# B&R Automation Studio project Parker_BMM_ST_V5_3147_V12 (part 8)

```c
		case 22000:
			pMold->Clamp.vRamp.Ts = tTask;
			pMold->Clamp.vRamp.Set = 0.0;

			/* call profile function */
			HydSCurveRamp(&pMold->Clamp.vRamp);

			pMold->Clamp.p_set = pMold->Clamp.p_old;
			pMold->Clamp.v_set = pMold->Clamp.vRamp.Out;

			if(pMold->Clamp.v_set < 0.1 && pMold->Clamp.v_set > -0.1)
			{
				pMold->Clamp.v_set = 0.0;
				pMold->Clamp.p_set =0;
				pMold->Clamp.Step = 0;
			}
			break;

		/* ----------------------------  Instance stop ------------------------- */
		case 30000:
			pMold->Clamp.Timer.IN      = 0;
			pMold->Clamp.LimitTimer.IN = 0;
			pMoldUser->Clamp.Timer.IN = 0;/*Albert*/

			pMold->ActInfo.ClampOpn = 0;
			pMold->ActInfo.ClampCls = 0;

			//*--VALVE_DIR--*//
			/*-- Close --*/
			pMold->ValveOut.ClampCls  = 0;
			pMold->ValveOut.ClampClsDiff = 0;
			pMold->ValveOut.ClampClsSlow = 0;
			/*-- Close_Tonnage_additional --*/
			pMold->ValveOut.Lock = 0;
			pMold->ValveOut.ClampClsAux = 0;

			/*-- Open --*/
			pMold->ValveOut.ClampOpn  = 0;
			pMold->ValveOut.ClampOpnDiff = 0;
			pMold->ValveOut.ClampOpnRelease = 0;

			//*--VALVE_PROP--*//
			pMold->ValveOut.ClampMoveValve = 0;

			/*-- Close --*/
			pMold->ValveOut.ClampClsDiff = 0;
			pMold->ValveOut.ClampClsSlow = 0;

			/*-- Open --*/
			pMold->ValveOut.ClampOpnDiff = 0;
			pMold->ValveOut.ClampOpnRelease = 0;

			pMold->Clamp.vRamp.Once = 0;
			pMold->Clamp.vRamp.Set = pMold->Clamp.v_set;

			pMold->Clamp.vRamp.Ts = tTask;

			pMold->Clamp.vRamp.Accel = INSTANCY_STOP_ACCEL;

			/* call profile function */
			HydSCurveRamp(&pMold->Clamp.vRamp);

			//	pMold->Clamp.p_set = 100.0;
			pMold->Clamp.v_set = pMold->Clamp.vRamp.Out;

			pMold->Clamp.Step = 31000;
			break;

		case 31000:
			pMold->Clamp.vRamp.Ts = tTask;
			pMold->Clamp.vRamp.Set = 0.0;

			/* call profile function */
			HydSCurveRamp(&pMold->Clamp.vRamp);

			pMold->Clamp.p_set = pMold->Clamp.p_old;
			pMold->Clamp.v_set = pMold->Clamp.vRamp.Out;

			if(pMold->Clamp.v_set < 0.1 && pMold->Clamp.v_set > -0.1)
			{
				pMold->Clamp.v_set = 0.0;
				pMold->Clamp.p_set =0;
				pMold->Clamp.Step = 0;
			}
			break;

		/* ----------------------------  Error step ------------------------- */
		case 40000:
			pMold->Clamp.Timer.IN      = 0;
			pMold->Clamp.LimitTimer.IN = 0;

			pMold->ActInfo.ClampOpn = 0;
			pMold->ActInfo.ClampCls = 0;

			pMold->Clamp.v_set = 0.0;
			pMold->Clamp.p_set =0;

			//*--VALVE_DIR--*//
			/*-- Close --*/
			pMold->ValveOut.ClampCls  = 0;
			pMold->ValveOut.ClampClsDiff = 0;
			pMold->ValveOut.ClampClsSlow = 0;
			/*-- Close_Tonnage_additional --*/
			pMold->ValveOut.Lock = 0;
			pMold->ValveOut.ClampClsAux = 0;

			/*-- Open --*/
			pMold->ValveOut.ClampOpn  = 0;
			pMold->ValveOut.ClampOpnDiff = 0;
			pMold->ValveOut.ClampOpnRelease = 0;

			//*--VALVE_PROP--*//
			pMold->ValveOut.ClampMoveValve = 0;

			/*-- Close --*/
			pMold->ValveOut.ClampClsDiff = 0;
			pMold->ValveOut.ClampClsSlow = 0;

			/*-- Open --*/
			pMold->ValveOut.ClampOpnDiff = 0;
			pMold->ValveOut.ClampOpnRelease = 0;

			break;

		/* ----------------------------  auto run stop ------------------------- */
		case 41000:
			pMold->Clamp.Timer.IN      = 0;
			pMold->Clamp.LimitTimer.IN = 0;

			pMold->ActInfo.ClampOpn = 0;
			pMold->ActInfo.ClampCls = 0;

			pMold->Clamp.Step = 42000;
			break;

		case 42000:
			pMold->Clamp.vRamp.Internal.Once = 0;
			pMold->Clamp.vRamp.Set = pMold->Clamp.v_set;

			pMold->Clamp.vRamp.Ts = tTask;

			pMold->Clamp.vRamp.Accel = INSTANCY_STOP_ACCEL;

			/* call profile function */
			HydSCurveRamp(&pMold->Clamp.vRamp);
			pMold->Clamp.Step = 43000;
			break;

		case 43000:
			pMold->Clamp.vRamp.Ts = tTask;
			pMold->Clamp.vRamp.Set = 0.0;

			/* call profile function */
			HydSCurveRamp(&pMold->Clamp.vRamp);

			//	pMold->Clamp.p_set = 100.0;
			pMold->Clamp.v_set = pMold->Clamp.vRamp.Out;

			if(pMold->Clamp.v_set < 0.1 && pMold->Clamp.v_set > -0.1)
			{
				pMold->Clamp.p_set =0;
				pMold->Clamp.v_set = 0.0;
				pMold->Clamp.Step = 40000;
			}
			break;
	}/* end of switch */

	if(pMold->Clamp.Step > 300 && pMold->Clamp.Step  < 800)
	{
		pMold->TimeDis.ClampClsAlarmTime = pMold->Clamp.LimitTimer.ET;
	}
	else if(pMold->Clamp.Step > 10300 && pMold->Clamp.Step  < 10800)
	{
		pMold->TimeDis.ClampOpnAlarmTime = pMold->Clamp.LimitTimer.ET;
	}

	/* ----------------- clamp open / close timeout --------------------  */
	if(1 == pMold->Clamp.LimitTimer.Q && 1 == gMachineInfo.TimeLimit)
	{
		if(pMold->Clamp.Step < 4000 && pMold->Clamp.Step > 200)		/* clamp close  */
		{
			pMold->Alarm.ClampNotAtClsDI = 1;
		}

		if(pMold->Clamp.Step < 13000 && pMold->Clamp.Step > 10200)	/* clamp open  */
		{
			pMold->Alarm.ClampNotAtOpnDI = 1;
		}

		pMold->Clamp.LimitTimer.IN = 0;
		pMold->Clamp.Step = 41000;
	}

	/* ----------------- clamp open / close action limit --------------------  */

	if(pMold->Clamp.Step < 3000 && pMold->Clamp.Step > 200) 	/* clamp close  */
	{

		if( 0 == pMold->TransDIn.SubMoldClsLimit)
		{
			pMold->Alarm.SubMoldNotAtOpnPos  = !pMold->TransDIn.SubMoldOpnLimit;
			pMold->Clamp.Step = 41000;
		}

		if( 0 == pMold->TransDIn.BottomSubMoldClsLimit)
		{
			pMold->Alarm.SubMoldNotAtOpnPos  = !pMold->TransDIn.BottomSubMoldClsLimit;
			pMold->Clamp.Step = 41000;
		}

		if(1 == gMachineInfo.Auto && 1 == gMachineFix.Option.bCoolPinUpNextCycClampCls)   /* 特殊模式  "於下一循環關模後轉一上"  */
		{
			//			if ( 0 == pMold->TransDIn.CoolPin2UpLimit || 0 == pMold->TransDIn.CoolPin3UpLimit )
			//			{
			//				pMold->Alarm.CoolPin2NotAtUpPos = !pMold->TransDIn.CoolPin2UpLimit;
			//				pMold->Alarm.CoolPin3NotAtUpPos	= !pMold->TransDIn.CoolPin3UpLimit;
			//				pMold->Clamp.Step = 41000;
			//			}
		}
		else
		{
			if (0 == pMold->TransDIn.CoolPinUpLimit )
			{
				pMold->Alarm.CoolPinNotAtUpPos	= !pMold->TransDIn.CoolPinUpLimit;
				pMold->Clamp.Step = 41000;
			}

		}

		if(0 == gMachineInfo.Auto)
		{
			if(0 == pMold->Robot.Transfer.BwPos)
			{
				pMold->Alarm.RobotNotAtBwPos = !pMold->Robot.Transfer.BwPos;
				pMold->Clamp.Step = 41000;
			}
		}

		if(1 == gMachineInfo.Auto )
		{
			if(0 == pMold->Carriage.FwPos)
			{
				pMold->Alarm.CarriageNotAtFwDI  = !pMold->Carriage.FwPos;
				pMold->Clamp.Step = 41000;
			}
		}

		/* 模内吹针在回位   */
		//      if(0 == pMold->TransDIn.InnerPinBwLimit)
		//      {
		//         pMold->Alarm.InnerPinNotAtBwPos = !pMold->TransDIn.InnerPinBwLimit;
		//         pMold->Clamp.Step = 41000;
		//      }

		//      if(1 == gMachineInfo.TimeLimit)
		//      {
		//         if(0 == pMold->Carriage.FwPos)
		//         {
		//            pMold->Alarm.CarriageNotAtFwDI  = !pMold->Carriage.FwPos;
		//            pMold->Clamp.Step = 41000;
		//         }
		//      }
		//      else
		//      {
		//         if(0 == pMold->Carriage.BwPos
		//			&& 0 == pMold->Carriage.FwPos
		//			&& 0 == pMold->BlowPin.UpPos)
		//         {
		//         	pMold->Alarm.CarriageNotAtBwDI = !pMold->Carriage.BwPos;
		//         	pMold->Alarm.BlowPinNotAtUpPos = !pMold->BlowPin.UpPos;
		//         	pMold->Clamp.Step = 41000;
		//         }
		//      }/* if(1 == gMachineInfo.Manual) */
	}/* if(pMold->Clamp.Step < 3000 && pMold->Clamp.Step > 200) */

	if(pMold->Clamp.Step < 13000 && pMold->Clamp.Step > 10200)  /* clamp open  */
	{

		/* 切飞边非退位  */
		if( 0 == pMold->TransDIn.TopDeflashBwLimit )
		{
			pMold->Alarm.TopDeflashNotAtBwPos = !pMold->TransDIn.TopDeflashBwLimit;
			pMold->Clamp.Step = 41000;
		}

		if( 0 == pMold->TransDIn.BottomDeflashBwLimit)
		{
			pMold->Alarm.BottomDeflashNotAtBwPos = !pMold->TransDIn.BottomDeflashBwLimit;
			pMold->Clamp.Step = 41000;
		}

		if(0 == gMachineInfo.Auto)
		{
			if(0 == pMold->TransDIn.ExtRobotUpLmit )
			{
				pMold->Alarm.ExtRobotNotAtUp = !pMold->TransDIn.ExtRobotUpLmit;
				pMold->Clamp.Step = 41000;
			}
		}

	}/* if(pMold->Clamp.Step < 13000 && pMold->Clamp.Step > 10200) */

	//	if((13000 >= pMold->Clamp.Step) && (10200 < pMold->Clamp.Step))
	//	{
	//		if(pMold == &RMold)
	//		{
	//			RobotClampTime.IN = pMold->Clamp.OpnPos;/*Albert RobotClampOpn*/
	//			RobotClampTime.PT = RobotClampTimePara;
	//		}
	//		if(pMold == & LMold)
	//		{
	//			LRobotClampTime.IN = pMold->Clamp.OpnPos;
	//			LRobotClampTime.PT = LRobotClampTimePara;
	//		}
	//	}
	//	else
	//	{
	////		RobotClampTime.IN = 0;/*Albert RobotClampOpn*/
	//	}
	//	if(pMold == &RMold)
	//	{
	//		if(RobotClampTime.Q)
	//		{
	//			RobotClampTime.IN = 0;
	//		}
	//		pMold->ValveOut.RobotClampOpn = RobotClampTime.Q;
	//
	//	}
	//	if(pMold == &LMold)
	//	{
	//		if(LRobotClampTime.Q)
	//		{
	//			LRobotClampTime.IN = 0;
	//		}
	//		pMold->ValveOut.RobotClampOpn = LRobotClampTime.Q;
	//	}

	/* ------------------------------------------------------------------------------ */
	/* ----------------- clamp output and proportional valve linear  ---------------- */
	/* ------------------------------------------------------------------------------ */

	if (pClampFix->eValveType == VALVE_PROP)
	{
		if(bClampPropValveOutputInverse == 0 )
		{
			if((pClampFix->Open.VoltageMax - pClampFix->Open.VoltageMin > 5.0) &&
				(pClampFix->Close.VoltageMin - pClampFix->Close.VoltageMax > 5.0))
			{
				pMold->Clamp.PropValveOk   = 1;
				pMold->Alarm.ClampValveErr = 0;
			}
			else
			{
				pMold->Clamp.PropValveOk   = 0;
				pMold->Alarm.ClampValveErr = 1;
			}
		}
		else
		{
			if((pClampFix->Open.VoltageMin - pClampFix->Open.VoltageMax > 5.0) &&
				(pClampFix->Close.VoltageMax - pClampFix->Close.VoltageMin > 5.0))
			{
				pMold->Clamp.PropValveOk   = 1;
				pMold->Alarm.ClampValveErr = 0;
			}
			else
			{
				pMold->Clamp.PropValveOk   = 0;
				pMold->Alarm.ClampValveErr = 1;
			}
		}

		pClampFix->Close.V_Max = 1000;
		pClampFix->Open.V_Max  = 1000;

		if(pMold->Clamp.v_set > pClampFix->Open.V_Max) pMold->Clamp.v_set = pClampFix->Open.V_Max;
		if(pMold->Clamp.v_set < -pClampFix->Close.V_Max) pMold->Clamp.v_set = -pClampFix->Close.V_Max;

		if(5000 == pMold->Clamp.Step || 15000 == pMold->Clamp.Step || 8500 == pMold->Clamp.Step)
		{
			if(bClampPropValveOutputInverse == 0)
			{
				pMold->Clamp.aoPropValve = pMold->Clamp.v_set * 32767/100;   /* 电压输出  0 -- 100 ---> 0.0 -- 10.0v*/
			}
			else
			{
				pMold->Clamp.aoPropValve = -(pMold->Clamp.v_set * 32767/100);   /* 电压输出  0 -- 100 ---> 0.0 -- 10.0v*/
			}

		}
		else
		{
			if(pMold->Clamp.v_set > 0 && pMold->Clamp.v_set <= pClampFix->Open.V_Max)
			{
				if(bClampPropValveOutputInverse == 0)
				{
					//Open +V
					pMold->Clamp.aoPropValve = 3276 * (pClampFix->Open.VoltageMin + pMold->Clamp.v_set/pClampFix->Open.V_Max *
						(pClampFix->Open.VoltageMax - pClampFix->Open.VoltageMin));
				}
				else
				{
					//Open -V
					pMold->Clamp.aoPropValve = 3276 * (pClampFix->Open.VoltageMin + (-pMold->Clamp.v_set/pClampFix->Open.V_Max) *
						(pClampFix->Open.VoltageMin - pClampFix->Open.VoltageMax));
				}
			}
			else if(pMold->Clamp.v_set < 0 && pMold->Clamp.v_set >= -pClampFix->Close.V_Max)
			{
				if(bClampPropValveOutputInverse == 0)
				{
					//Close -V
					pMold->Clamp.aoPropValve = 3276 * (pClampFix->Close.VoltageMin + pMold->Clamp.v_set/pClampFix->Close.V_Max *
						(pClampFix->Close.VoltageMin - pClampFix->Close.VoltageMax));
				}
				else
				{
					//Close +V
					pMold->Clamp.aoPropValve = 3276 * (pClampFix->Close.VoltageMin + (-pMold->Clamp.v_set/pClampFix->Open.V_Max) *
						(pClampFix->Close.VoltageMax - pClampFix->Close.VoltageMin));
				}
			}
			else
			{
				pMold->Clamp.aoPropValve = 0;
			}
		}
	}
	else
	{
		pMold->Alarm.ClampValveErr = 0;
	}

}/*end of function */

void ClampDriveToggle_Drive(Mold_typ * pMold, Clamp_Fix_typ * pClampFix,Clamp_Para_typ * pClampPara,SPC_Mold_typ * pSPC, Mold_Para_User_typ * pMoldUser)
{
	/*  pMax set  */
	if(pMold == & LMold)
	{
		pClampFix->pMax = 100;
	}
	else
	{
		pClampFix->pMax = 100;
	}

	if(1 == gMachineOut.OilPump)
	{
		if(tErrorDelay >= tTask)tErrorDelay = tErrorDelay - tTask;
		if(tErrorDelay < tTask)
		{
			if(pMold == & LMold)
			{
				LMold.HwAlarm.ClampNetworkErr = !LMold.Clamp.NetworkInit;
				LMold.HwAlarm.ClampPowerOn    = !LMold.Clamp.PowerOn;
			}
			else
			{
				RMold.HwAlarm.ClampNetworkErr = !RMold.Clamp.NetworkInit;
				RMold.HwAlarm.ClampPowerOn    = !RMold.Clamp.PowerOn;
			}
		}

		if((RMold.HwAlarm.ClampNetworkErr ||RMold.HwAlarm.ClampPowerOn)||(LMold.HwAlarm.ClampNetworkErr ||LMold.HwAlarm.ClampPowerOn))
		{
			gMachineOut.OilPump = 0;
			gPROCESS_info.oilpumpStop = 1;   //request manual mode
		}
	}
	else
	{
		tErrorDelay = 0.1;
		if(pMold == & LMold)
		{
			//			LMold.HwAlarm.ClampNetworkErr = 0;
			//			LMold.HwAlarm.ClampPowerOn    = 0;
		}
		else
		{
			//			RMold.HwAlarm.ClampNetworkErr = 0;
			//			RMold.HwAlarm.ClampPowerOn    = 0;
		}
	}

	/* ------------- clamp axis alarms ------------- */

	pMold->HwAlarm.ClampAxisErr    = pMold->Clamp.Error;

   /*********************************************************************************
  	**                            HMI data value to PLC                             **
  	*********************************************************************************/
	if(pClampFix->Length < 100.0)pClampFix->Length = 320.0;
	if(pClampFix->Tolerance < 0.1)pClampFix->Tolerance = 0.1;

	if(pClampFix->Close.V_Max < 500.0)pClampFix->Close.V_Max = 1000.0;
	if(pClampFix->Open.V_Max  < 500.0)pClampFix->Open.V_Max  = 1000.0;

	if(pClampFix->Close.VoltageMax > -3.0)pClampFix->Close.VoltageMax = -10.0;
	if(pClampFix->Open.VoltageMax  < 3.0 )pClampFix->Open.VoltageMax  = 10.0;

	if(pClampFix->pPress2Hold  < 10 )pClampFix->pPress2Hold  = 10.0;
	if(pClampFix->pPress2Hold  > 70 )pClampFix->pPress2Hold  = 70;

	pMold->Clamp.Tolerance = pClampFix->Tolerance;

	pMold->Clamp.S_Cls = pClampPara->S_Cls;
	pMold->Clamp.S_ClsEnd = pClampPara->S_ClsEnd;

	pMold->Clamp.S_CutterCls = pClampPara->S_CutterCls;
	pMold->Clamp.S_BlowPinUp = pClampPara->S_BlowPinUp;

	pMold->Clamp.V_Cls = pClampPara->V_Cls * pClampFix->Close.V_Max /100.0;
	pMold->Clamp.V_ClsSlow = pClampPara->V_ClsSlow * pClampFix->Close.V_Max /100.0;
	pMold->Clamp.V_Tonnage = pClampPara->V_Tonnage * pClampFix->Close.V_Max /100.0;
	pMold->Clamp.V_ClsLock = pClampPara->V_Lock * pClampFix->Close.V_Max/100.0;/*2018.7.17 Albert */

	pMold->Clamp.P_Cls		= pClampPara->P_Cls 	= 100;
	pMold->Clamp.P_ClsSlow	= pClampPara->P_ClsSlow = 100;
	pMold->Clamp.P_Tonnage	= pClampPara->P_Tonnage;
	pMold->Clamp.P_Lock		= pClampPara->P_Lock;

	pMold->Clamp.S_OpnSlow2   = pClampPara->S_OpnSlow2;
	pMold->Clamp.S_OpnSlow    = pClampPara->S_OpnSlow;
	pMold->Clamp.S_OpnEnd     = pClampPara->S_OpnEnd;

	pMold->Clamp.S_ScrewBw    = pClampPara->S_ScrewBw;
	pMold->Clamp.S_SubMoldOut = pClampPara->S_SubMoldOut;

	if(	pClampPara->S_SubMoldIn <= pClampPara->S_OpnSlow2)	pClampPara->S_SubMoldIn   = pClampPara->S_OpnSlow2;
	if(	pClampPara->S_SubMoldIn >= pClampPara->S_OpnEnd)	pClampPara->S_SubMoldIn   = pClampPara->S_OpnEnd;
	pMold->Clamp.S_SubMoldIn   = pClampPara->S_SubMoldIn;

	pMold->Clamp.V_Opn = pClampPara->V_Opn * pClampFix->Open.V_Max /100.0;
	pMold->Clamp.V_OpnSlow = pClampPara->V_OpnSlow * pClampFix->Open.V_Max /100.0;
	pMold->Clamp.V_OpnSlow2 = pClampPara->V_OpnSlow2 * pClampFix->Open.V_Max /100.0;

	pMold->Clamp.P_Opn		= pClampPara->P_Opn			= 100;
	pMold->Clamp.P_OpnSlow	= pClampPara->P_OpnSlow 	= 100;
	pMold->Clamp.P_OpnSlow2	= pClampPara->P_OpnSlow2	= 100;

	if(0 == pClampPara->V_OpnReset)pClampPara->V_OpnReset = 2.0;
	pMold->Clamp.V_OpnReset = pClampPara->V_OpnReset * pClampFix->Open.V_Max /100.0;
	pClampPara->P_OpnReset	= 100;

	if(pClampFix->Open.accel_stop < 100)pClampFix->Open.accel_stop = INSTANCY_STOP_DECEL;
	if(pClampFix->Close.accel_stop < 100)pClampFix->Close.accel_stop = INSTANCY_STOP_DECEL;
	/*********************************************************************************
  	**                            linear calibration status                        **
  	*********************************************************************************/
  	/* get calibration data  */
	if(pClampFix->Max < pClampFix->Zero)
	{
		pMold->Clamp.ZeroPos = pClampFix->Max;
		pMold->Clamp.MaxPos = pClampFix->Zero;
	}
	else
	{
		pMold->Clamp.MaxPos  = pClampFix->Max;
		pMold->Clamp.ZeroPos = pClampFix->Zero;
	}

	if(pMold->Clamp.ZeroPos != 0                           &&
		pMold->Clamp.MaxPos > (pMold->Clamp.ZeroPos + 10000) &&
		pMold->Clamp.As     > (pMold->Clamp.ZeroPos - 5000 ) &&
		pMold->Clamp.As     < (pMold->Clamp.MaxPos  + 2000 ))
	{
		pMold->Clamp.CalOK = pMold->Clamp.NetworkInit;
	}
	else
	{
		pMold->Clamp.CalOK = 0;
	}

	pClampFix->CalibOK = pMold->Clamp.CalOK;

	if(1 == pMold->Clamp.CalOK)
	{
		if(pClampFix->Max < pClampFix->Zero)
		{
			pMold->Clamp.mmAsDrive = 1.0 *(pMold->Clamp.MaxPos - pMold->Clamp.As) * pClampFix->Length /
				(pMold->Clamp.MaxPos - pMold->Clamp.ZeroPos);

			pMold->Clamp.mmDriveTonnage = 1.0 *(pMold->Clamp.MaxPos - pClampFix->ecMaxForce) * pClampFix->Length /
				(pMold->Clamp.MaxPos - pMold->Clamp.ZeroPos);

			if(pMold->Clamp.mmDriveTonnage > 20 || pMold->Clamp.mmDriveTonnage < -20)
			{
				pMold->Clamp.mmDriveTonnage = 0.0;
			}
		}
		else
		{
			pMold->Clamp.mmAsDrive = 1.0 *(pMold->Clamp.As - pMold->Clamp.ZeroPos) * pClampFix->Length /
				(pMold->Clamp.MaxPos - pMold->Clamp.ZeroPos);

			pMold->Clamp.mmDriveTonnage = 1.0 *(pClampFix->ecMaxForce - pMold->Clamp.ZeroPos) * pClampFix->Length /
				(pMold->Clamp.MaxPos - pMold->Clamp.ZeroPos);

			if(pMold->Clamp.mmDriveTonnage > 20 || pMold->Clamp.mmDriveTonnage < -20)
			{
				pMold->Clamp.mmDriveTonnage = 0.0;
			}
		}
	}
	else
	{
		pMold->Clamp.mmAsDrive = pMold->Clamp.mmAsDrive;

		if(0 == gMachineInfo.Calib)	/* 非调校模式  */
		{
			if(pMold->Clamp.Step > 0 && pMold->Clamp.Step < 20000)
			{
				pMold->Clamp.Step = 0;
				pMold->Alarm.ClampCalErr = 1;
			}
		}
	}/* if(1 == pMold->Clamp.CalOK) */

	/*  toggle clamp linear  */
	pClampFix->ToggleLin[0].X = 0.0;
	pClampFix->ToggleLin[0].Y = 0.0;

	pClampFix->ToggleLin[ToggleLinNodeNum-1].X = pClampFix->Length;
	pClampFix->ToggleLin[ToggleLinNodeNum-1].Y = pClampFix->Length;

	if(pMold == &LMold)
	{
		TogLinearL.Y = pMold->Clamp.mmAsDrive;
		HydLinear(&TogLinearL);

		if(TogLinearL.status != 0)
		{
			pMold->Alarm.ClampLinNotOK = 1;
			pMold->Clamp.mmAs = pMold->Clamp.mmAsDrive;
		}
		else
		{
			pMold->Clamp.mmAs = TogLinearL.X;
		}

		//		if(pMold->Clamp.As < pMold->Clamp.ZeroPos)
		//		{
		//			pMold->Clamp.mmAs = pMold->Clamp.mmAsDrive;
		//		}
	}
	else if(pMold == &RMold)
	{
		TogLinearR.Y = pMold->Clamp.mmAsDrive;
		HydLinear(&TogLinearR);

		if(TogLinearR.status != 0)
		{
			pMold->Alarm.ClampLinNotOK = 1;
			pMold->Clamp.mmAs = pMold->Clamp.mmAsDrive;
		}
		else
		{
			pMold->Clamp.mmAs = TogLinearR.X;
		}

		//		if(pMold->Clamp.As < pMold->Clamp.ZeroPos)
		//		{
		//			pMold->Clamp.mmAs = pMold->Clamp.mmAsDrive;
		//		}
	}

	/*  relative position  */
	pMold->Clamp.Ss = pMold->Clamp.As;
	pMold->Clamp.mmAsMax = pClampFix->Length + 10;

	/* gAlarm time value    */
	if(!pMold->TimeSet.ClampOpnAlarmTime)pMold->TimeSet.ClampOpnAlarmTime = 1000;  /* 10s  */
	if(!pMold->TimeSet.ClampClsAlarmTime)pMold->TimeSet.ClampClsAlarmTime = 1000;  /* 10s  */

	/* clamp open or close position flag  */
	pMold->Clamp.ClsPos = pMold->TransDIn.ClampClsLimit &&
		(pMold->Clamp.mmAs < (pMold->Clamp.S_ClsEnd + pMold->Clamp.Tolerance));
	pMold->Clamp.OpnPos = pMold->TransDIn.ClampOpnLimit &&
		(pMold->Clamp.mmAs > (pMold->Clamp.S_OpnEnd - pMold->Clamp.Tolerance));

	pMold->Clamp.OpnOverHalf = pMold->Clamp.mmAs >= pClampPara->S_SubMoldOut;

	if(pMold->Clamp.mmAsDrive > pMold->Clamp.mmDriveTonnage - 0.03 && pMold->Clamp.mmAsDrive < pMold->Clamp.mmDriveTonnage + 0.03)
	{
		pMold->Clamp.TonnagePos = 1;
	}
	else
	{
		pMold->Clamp.TonnagePos = 0;
	}

	/* ------------------ function current position ------------------ */
	pMold->Clamp.vProfGen.s_act = pMold->Clamp.mmAsDrive;
	pMold->Clamp.vProfGen.v_act = pMold->Clamp.v_act; // mmAsDrive -> v_act

	/* clamp open or close step  */
	switch ( pMold->Clamp.Step )
	{
		/*------------------ stop all the output ------------------*/
		case 0:
			pMold->Clamp.v_set = 0;
			pMold->Clamp.p_set = 0;

			pMold->ActInfo.ClampOpn  = 0;
			pMold->ActInfo.ClampCls  = 0;

			pMold->Clamp.Timer.IN	   = 0;
			pMold->Clamp.LimitTimer.IN = 0;

			break;
		/*------------------ Clean Valve ------------------*/
		case 5:
			/*Clean Valve*/
			break;
		/*--------------------------------------------------------------- */
		/*------------------------ Clamp close -------------------------- */
		/*--------------------------------------------------------------- */
		case 100: /* close delay*/
			if(pMold->TimeSet.ClampClsDelay != 0)
			{
				pMold->Clamp.Timer.IN = 1;
				pMold->Clamp.Timer.PT = pMold->TimeSet.ClampClsDelay;

				//gExSPC
				if(pMold == & LMold)
				{
					gExSPC[ExIndex].LMold.ClampClsDelay = pMold->TimeSet.ClampClsDelay/100.0;
				}
				else
				{
					gExSPC[ExIndex].RMold.ClampClsDelay = pMold->TimeSet.ClampClsDelay/100.0;
				}
				//				pMold->TimeDis.ClampClsDelay = 0;
				pMold->Clamp.Step = 200;
			}
			else
			{
				pMold->Clamp.Step = 300;
			}
			break;

		case 200: /* delay ok */
			pMold->TimeDis.ClampClsDelay = pMold->Clamp.Timer.ET;
			if (1 == pMold->Clamp.Timer.Q)
			{
				pMold->Clamp.Timer.IN        = 0;
				//				pMold->TimeDis.ClampClsDelay = 0;
				pMold->Clamp.Step = 300;
			}
			break;

		case 300:	/* time limit  */
			if(0 == pMold->Clamp.ClsHWSwitch)
			{
				if(pMold == &LMold)
				{
					pMold->Clamp.S_ClsDrive  = xTogLinearLTrans(pClampPara->S_Cls);
					pMold->Clamp.S_ClsEndDrive = xTogLinearLTrans(pClampPara->S_ClsEnd);
				}
				else
				{
					pMold->Clamp.S_ClsDrive  = xTogLinearRTrans(pClampPara->S_Cls);
					pMold->Clamp.S_ClsEndDrive = xTogLinearRTrans(pClampPara->S_ClsEnd);
				}

				pMold->Clamp.LimitTimer.IN = 1;
				pMold->Clamp.LimitTimer.PT = pMold->TimeSet.ClampClsAlarmTime;

				pMold->Clamp.vProfGen.Ts = tTask;
				pMold->Clamp.vProfGen.Tj = pClampFix->Close.Tj;
				pMold->Clamp.vProfGen.Td = pClampFix->Close.Td;

				pMold->Clamp.vProfGen.accel = pClampFix->Close.accel;
				if(pMold->Clamp.vProfGen.accel <= 0.0)pMold->Clamp.vProfGen.accel = 1000;

				pMold->Clamp.vProfGen.decel = pClampFix->Close.accel;
				if(pMold->Clamp.vProfGen.decel <= 0.0)pMold->Clamp.vProfGen.decel = 1000;

				pMold->Clamp.vProfGen.decel_end = pClampFix->Close.decel_end;
				if(pMold->Clamp.vProfGen.decel_end <= 0.0)pMold->Clamp.vProfGen.decel_end = 100;

				pMold->Clamp.vProfGen.v_start = 0.0;

				if (pMold->Clamp.S_Cls >0) //close quick
				{
					//					pMold->Clamp.vProfGen.v_end	= pMold->Clamp.V_ClsSlow;
					//					pMold->Clamp.vProfGen.s_end = pMold->Clamp.S_ClsDrive;
					//					pMold->Clamp.vProfGen.init  = 1;

					if(pMold->TimeSet.ClampLockTime == 0 || 1 == gMachineInfo.Manual )
					{
						pMold->Clamp.vProfGen.v_end = 0;
//						pMold->Clamp.vProfGen.v_end	= pMold->Clamp.V_Tonnage/2;
					}
					else
					{
						pMold->Clamp.vProfGen.v_end = 0;
//						pMold->Clamp.vProfGen.v_end	= pMold->Clamp.V_Tonnage/2;
					}
					pMold->Clamp.vProfGen.s_end = pMold->Clamp.S_ClsEndDrive;
					pMold->Clamp.vProfGen.init  = 1;

					pMold->Clamp.Step = 400;
				}
				else   							//close slow
				{
					if(pMold->TimeSet.ClampLockTime == 0 || 1 == gMachineInfo.Manual )
					{
						pMold->Clamp.vProfGen.v_end = 0;
//						pMold->Clamp.vProfGen.v_end	= pMold->Clamp.V_Tonnage/2;
					}
					else
					{
						pMold->Clamp.vProfGen.v_end = 0;
//						pMold->Clamp.vProfGen.v_end	= pMold->Clamp.V_Tonnage/2;
					}
					pMold->Clamp.vProfGen.s_end = pMold->Clamp.S_ClsEndDrive;
					pMold->Clamp.vProfGen.init  = 1;

					pMold->Clamp.Step = 500;
				}

			}
			else
			{
				pMold->HwAlarm.ClampClsHWSwitch = 1;
				pMold->Clamp.Step = 41000;
			}
			break;

		case 400:	/* close quick  */
			pMold->ActInfo.ClampCls  = 1;

			pMold->Clamp.vProfGen.v_set = pMold->Clamp.V_Cls;
			/* call profile function */
			HydvProfGen(& pMold->Clamp.vProfGen);

			pMold->Clamp.p_set = pClampPara->P_Cls = 100.0;
			pMold->Clamp.v_set = pMold->Clamp.vProfGen.v_out;

			pMold->Clamp.actTjCls = pMold->Clamp.vProfGen.Tj;

			/*  reached target position */
			if(pMold->Clamp.vProfGen.s_act <= pMold->Clamp.S_ClsDrive)
			{
				//				pMold->Clamp.vProfGen.v_start = pMold->Clamp.v_set;
				//				if(pMold->TimeSet.ClampLockTime == 0 || 1 == gMachineInfo.Manual )
				//				{
				//					pMold->Clamp.vProfGen.v_end = 0;
				//				}
				//				else
				//				{
				//					pMold->Clamp.vProfGen.v_end	= pMold->Clamp.V_Tonnage/2;
				//				}
				//				pMold->Clamp.vProfGen.s_end = pMold->Clamp.S_ClsEndDrive;
				//				pMold->Clamp.vProfGen.init  = 1;

				pMold->Clamp.Step = 500;
			}

			if(1 == pMold->Clamp.ClsHWSwitch)
			{
				pMold->HwAlarm.ClampClsHWSwitch = 1;
				pMold->Clamp.Step = 41000;
			}
			break;

		case 500:	/* close slow  */

			pMold->ActInfo.ClampCls  = 1;

			pMold->Clamp.vProfGen.v_set = pMold->Clamp.V_ClsSlow;

			/* call profile function */
			HydvProfGen(& pMold->Clamp.vProfGen);

			pMold->Clamp.p_set = pClampPara->P_ClsSlow;
			pMold->Clamp.v_set = pMold->Clamp.vProfGen.v_out;

			/*  reached target position */
			if(pMold->Clamp.vProfGen.s_act <= pMold->Clamp.vProfGen.s_end + pMold->Clamp.Tolerance)
			{
				pMold->Clamp.v_set = 0;
				pMold->Clamp.LimitTimer.IN = 0;
				if(gMachineInfo.Manual)
				{
					pMold->Clamp.Step = 3400;
				}
				else if(gMachineInfo.Auto)
				{
					pMold->Clamp.Step = 600;
				}
			}

			if(1 == pMold->Clamp.ClsHWSwitch)
			{
				pMold->HwAlarm.ClampClsHWSwitch = 1;
				pMold->Clamp.Step = 41000;
			}
			break;

		case 600:
			pMold->ActInfo.ClampOpn  = 0;
			pMold->ActInfo.ClampCls  = 0;

			pMold->Clamp.p_set = 0;
			pMold->Clamp.v_set = 0;

			pMold->Clamp.Timer.IN = 0;
			pMold->Clamp.LimitTimer.IN = 0;
			pMoldUser->Clamp.Timer.IN = 0;

			if(1 == gMachineInfo.Auto)
			{
				pSPC->tCalmpCls = pMold->Clamp.LimitTimer.ET/100.0;
				pMold->Clamp.Step = 3000;

				//gExSPC
				if(pMold == & LMold)
				{
					gExSPC[ExIndex].LMold.tCalmpCls = pMold->Clamp.LimitTimer.ET/100.0;
				}
				else
				{
					gExSPC[ExIndex].RMold.tCalmpCls = pMold->Clamp.LimitTimer.ET/100.0;
				}

			}
			else
			{
				pMold->Clamp.Step = 3000;
			}
			break;

		/* lock Start （加壓）*/
		/*---------*/
		case 3400:
			/*---------*/
			//lock
			if(pMold->TimeSet.ClampLockTime != 0)
			{
				pMold->ActInfo.ClampOpn  = 0;
				pMold->ActInfo.ClampCls  = 1;

				pMold->Clamp.Timer.IN = 1;
				pMold->Clamp.Timer.PT = pMold->TimeSet.ClampLockTime;

				pMold->Clamp.vTimeProf.Ts = tTask;
				pMold->Clamp.vTimeProf.t_move = pMold->TimeSet.ClampLockTime * 0.01;

				pMold->Clamp.vTimeProf.v_set   = pMold->Clamp.V_Tonnage;
				pMold->Clamp.vTimeProf.v_start = pMold->Clamp.v_set;
				pMold->Clamp.vTimeProf.v_end   = 0.0;

				pMold->Clamp.vTimeProf.accel = 1000;
				if(pMold->Clamp.vTimeProf.accel <= 0.0)pMold->Clamp.vTimeProf.accel = 1000;

				pMold->Clamp.vTimeProf.decel = 1000;
				if(pMold->Clamp.vTimeProf.decel <= 0.0)pMold->Clamp.vTimeProf.decel = 1000;

				pMold->Clamp.vTimeProf.init = 1;
				pMold->Clamp.Step = 3500;
			}
			else
			{
				pMold->Clamp.Step = 3800;  //3900
			}
			break;

		/*---------*/
		case 3500:	 /*(Press torque procedure)*/
			/*---------*/

			pMold->ActInfo.ClampCls  = 1;

			HydvTimeProf(&pMold->Clamp.vTimeProf);

			pMold->Clamp.p_set = pMold->Clamp.P_Tonnage;
			pMold->Clamp.v_set = -pMold->Clamp.vTimeProf.v_out;

			pMold->TimeDis.ClampLockTime = pMold->Clamp.Timer.ET;
			if (1 == pMold->Clamp.Timer.Q)
			{
//				pMold->Clamp.v_set = 0;
				pMold->Clamp.Timer.IN      = 0;
				pMold->Clamp.Step = 3600;
			}

//			pMold->TimeDis.ClampClsAlarmTime = pMold->Clamp.LimitTimer.ET;

			if(1 == pMold->Clamp.ClsHWSwitch)
			{
				pMold->HwAlarm.ClampClsHWSwitch = 1;
				pMold->Clamp.Step = 41000;
			}
			break;

		/*  --------------------------------------------------------------- */
		/*  -------------- Press torque 2 procedure Set ------------------- */
		case 3600:	/*(Press torque 2 procedure Set)*/
			/*---------*/
			//lock
			if(pMold->TimeSet.ClampLockTime != 0)
			{
				pMold->ActInfo.ClampOpn  = 0;
				pMold->ActInfo.ClampCls  = 1;

				pMold->Clamp.Timer.IN = 1;
				pMold->Clamp.Timer.PT = pMold->TimeSet.ClampClsPress2HoldTime;

				pMold->Clamp.vTimeProf.Ts = tTask;
				pMold->Clamp.vTimeProf.t_move = pMold->TimeSet.ClampClsPress2HoldTime * 0.01;

				pMold->Clamp.vTimeProf.v_set   = pMold->Clamp.V_Tonnage;
				pMold->Clamp.vTimeProf.v_start = pMold->Clamp.v_set;
				pMold->Clamp.vTimeProf.v_end   = 0.0;

				pMold->Clamp.vTimeProf.accel = Test_vTimeProf_accel;
				if(pMold->Clamp.vTimeProf.accel <= 0.0)pMold->Clamp.vTimeProf.accel = 1000;

				pMold->Clamp.vTimeProf.decel = Test_vTimeProf_decel;
				if(pMold->Clamp.vTimeProf.decel <= 0.0)pMold->Clamp.vTimeProf.decel = 1000;

				pMold->Clamp.vTimeProf.init = 1;
				pMold->Clamp.Step = 3700;
			}
			else
			{
				pMold->Clamp.Step = 3800;  //3900
			}
			break;

		/*---------*/
		case 3700:	 /*(Press torque 2 procedure)*/
		/*---------*/

			pMold->ActInfo.ClampCls  = 1;

			pMold->TimeDis.ClampClsPress2HoldTime = pMold->Clamp.Timer.ET;
			HydvTimeProf(&pMold->Clamp.vTimeProf);

			pMold->Clamp.p_set = pClampFix->pPress2Hold;
			pMold->Clamp.v_set = -pMold->Clamp.vTimeProf.v_out;

//			pMold->TimeDis.ClampLockTime = pMold->Clamp.Timer.ET;
			if (1 == pMold->Clamp.Timer.Q)
			{
				pMold->Clamp.v_set = 0;
				pMold->Clamp.Timer.IN      = 0;
				pMold->Clamp.Step = 3800;
			}

//			pMold->TimeDis.ClampClsAlarmTime = pMold->Clamp.LimitTimer.ET;

			if(1 == pMold->Clamp.OpnHWSwitch)
			{
				pMold->HwAlarm.ClampOpnHWSwitch = 1;
				pMold->Clamp.Step 	= 41000;
			}
			else if(1 == pMold->Clamp.ClsHWSwitch)
			{
				pMold->HwAlarm.ClampClsHWSwitch = 1;
				pMold->Clamp.Step 	= 41000;
			}
			break;

		case 3800: //End
			pMold->ActInfo.ClampCls  = 0;
			pMold->ActInfo.ClampOpn  = 0;

			pMold->Clamp.Timer.IN   = 0;
			pMold->Clamp.LimitTimer.IN = 0;

			pMold->Clamp.v_set = 0;

			pMold->Clamp.Step = 3900;
			break;

		case 3000:
			RobotClampTime.IN = 0;
			LRobotClampTime.IN = 0;
			break;

		case 3900:

			RobotClampTime.IN = 0;
			LRobotClampTime.IN = 0;
			break;

		/* --------------- 调校关模 --------------- */
		case 5000:
			if(0 == pMold->Clamp.ClsHWSwitch)
			{
				pMold->ActInfo.ClampCls  = 1;

				pMold->Clamp.p_set = pClampFix->pCalibZero;
				pMold->Clamp.v_set = -pClampFix->vCalibZero*10;
			}

			if(1 == pMold->Clamp.ClsHWSwitch)
			{
				pMold->HwAlarm.ClampClsHWSwitch = 1;
				pMold->Clamp.Step = 41000;
			}
			break;
		/* --------------- 绞牙微开模 --------------- */
		case 11100:
			if(1 == pMold->Option.Screw)
			{
				pMold->Clamp.LimitTimer.IN = 1;
				pMold->Clamp.LimitTimer.PT = pMold->TimeSet.ClampOpnAlarmTime;

				pMold->Clamp.vProfGen.Ts = tTask;
				pMold->Clamp.vProfGen.Tj = pClampFix->Open.Tj;
				pMold->Clamp.vProfGen.Td = pClampFix->Open.Td;

				pMold->Clamp.vProfGen.accel = pClampFix->Open.accel;
				if(pMold->Clamp.vProfGen.accel <= 0.0)pMold->Clamp.vProfGen.accel = 1000;

				pMold->Clamp.vProfGen.decel = pClampFix->Open.accel;
				if(pMold->Clamp.vProfGen.decel <= 0.0)pMold->Clamp.vProfGen.decel = 1000;

				pMold->Clamp.vProfGen.decel_end = pClampFix->Open.decel_end;
				if(pMold->Clamp.vProfGen.decel_end <= 0.0)pMold->Clamp.vProfGen.decel_end = 100;

				pMold->Clamp.vProfGen.v_start = 0.0;
				pMold->Clamp.vProfGen.v_end	= 0.0;
				pMold->Clamp.vProfGen.s_end = pMold->Clamp.S_ScrewBw;
				pMold->Clamp.vProfGen.init  = 1;

				pMold->Clamp.Step = 11200;
			}
			else
			{
				pMold->Clamp.Step = 13000;
			}
			break;

		case 11200:
			pMold->ActInfo.ClampOpn  = 1;

			pMold->Clamp.vProfGen.v_set = pMold->Clamp.V_OpnSlow;

			/* call profile function */
			HydvProfGen(& pMold->Clamp.vProfGen);

			pMold->Clamp.p_set = pClampPara->P_OpnSlow;
			pMold->Clamp.v_set = pMold->Clamp.vProfGen.v_out;

			pMold->Clamp.actTjOpn = pMold->Clamp.vProfGen.Tj;

			/*  reached target position */
			if(pMold->Clamp.mmAs > pMold->Clamp.S_ScrewBw)
			{
				pMold->ActInfo.ClampOpn  = 0;

				pMold->Clamp.v_set = 0;
				pMold->Clamp.Step = 11300;
			}
			if(1 == pMold->Clamp.OpnHWSwitch)
			{
				pMold->HwAlarm.ClampOpnHWSwitch = 1;
				pMold->Clamp.Step = 41000;
			}
			break;

		case 11300:
			pMold->Clamp.LimitTimer.IN = 0;

			pMold->Clamp.v_set  = 0;
			pMold->Clamp.p_set =0;
			pMold->ActInfo.ClampOpn  = 0;

			pMold->Clamp.Step = 13000;
			break;

		/*-------------------------------------------------------------------------------*/
		/*----------------------- 開模洩壓 + 子模微開模 ---------------------------------*/
		/*-------------------------------------------------------------------------------*/
		case 12100:/*UnLock Process   開模洩壓*/
			//			if(pMoldUser->TimeSet.ClampUnLockTime != 0)
			//			{
			//				pMold->Clamp.Timer.IN = 1;
			//				pMold->Clamp.Timer.PT = pMoldUser->TimeSet.ClampUnLockTime;
			//				pMold->Clamp.Step 	  = 12110;
			//			}
			//			else
			//			{
			if( 1 == pMold->Option.SubMold)
			{
				pMold->Clamp.Step = 12130; //微開延遲+ 微開
			}
			else
			{
				pMold->Clamp.Step = 12300; //微開延遲+ 微開 跳過
			}

			//			}
			break;

		//		case 12110:/*Wait UnLock Finish*/
		//			pMoldUser->TimeDis.ClampUnLockTime = pMold->Clamp.Timer.ET;
		//			if(pMold->Clamp.Timer.Q)
		//			{
		//				pMold->Clamp.Timer.IN = 0;
		//				//				pMold->Clamp.Step = 12130;  // 微開模延遲不使用
		//				pMold->Clamp.Step = 12150;
		//			}
		//			break;

		case 12130: /* open delay */
			if(pMold->TimeSet.ClampMircoOpnDelay != 0)
			{
				pMold->Clamp.Timer.IN = 1;
				pMold->Clamp.Timer.PT = pMold->TimeSet.ClampMircoOpnDelay;
				pMold->Clamp.Step 	  = 12140;
			}
			else
			{
				pMold->Clamp.Step = 12150;
			}
			break;

		case 12140: /* delay ok 微開模*/
			pMold->TimeDis.ClampMircoOpnDelay = pMold->Clamp.Timer.ET;
			if (1 == pMold->Clamp.Timer.Q)
			{
				pMold->Clamp.Timer.IN        = 0;
				pMold->Clamp.Step = 12150;
			}
			break;

		case 12150:
			pMold->Clamp.LimitTimer.IN = 1;
			pMold->Clamp.LimitTimer.PT = pMold->TimeSet.ClampOpnAlarmTime;

			pMold->Clamp.vProfGen.Ts = tTask;
			pMold->Clamp.vProfGen.Tj = pClampFix->Open.Tj;
			pMold->Clamp.vProfGen.Td = pClampFix->Open.Td;

			pMold->Clamp.vProfGen.accel = pClampFix->Open.accel;
			if(pMold->Clamp.vProfGen.accel <= 0.0)pMold->Clamp.vProfGen.accel = 1000;

			pMold->Clamp.vProfGen.decel = pClampFix->Open.accel;
			if(pMold->Clamp.vProfGen.decel <= 0.0)pMold->Clamp.vProfGen.decel = 1000;

			pMold->Clamp.vProfGen.decel_end = pClampFix->Open.decel_end;
			if(pMold->Clamp.vProfGen.decel_end <= 0.0)pMold->Clamp.vProfGen.decel_end = 100;

			pMold->Clamp.vProfGen.v_start = 0.0;
			pMold->Clamp.vProfGen.v_end	= 0.0;

			pMold->Clamp.vProfGen.s_end = pMold->Clamp.S_SubMoldOut; // 微開模

			pMold->Clamp.vProfGen.init  = 1;

			pMold->Clamp.Step = 12200;
			break;

		case 12200:		/* 開到 微開模 位置*/

			pMold->ActInfo.ClampOpn  = 1;

			pMold->Clamp.vProfGen.v_set = pMold->Clamp.V_OpnSlow;

			/* call profile function */
			HydvProfGen(& pMold->Clamp.vProfGen);

			pMold->Clamp.p_set = pClampPara->P_OpnSlow;
			pMold->Clamp.v_set = pMold->Clamp.vProfGen.v_out;

			pMold->Clamp.actTjOpn = pMold->Clamp.vProfGen.Tj;

			/*  reached target position */

			if(pMold->Clamp.mmAs > pMold->Clamp.S_SubMoldOut - 0.1)  // 微開模
			{
				pMold->Clamp.v_set  = 0;
				pMold->Clamp.p_set  = 0;
				pMold->Clamp.Step = 12300;
			}

			if(1 == pMold->Clamp.OpnHWSwitch)
			{
				pMold->HwAlarm.ClampOpnHWSwitch = 1;
				pMold->Clamp.Step = 41000;
			}
			break;

		case 12300:
			pMold->Clamp.LimitTimer.IN = 0;
			pMold->Clamp.Timer.IN = 0;
			pMold->ActInfo.ClampOpn  = 0;
			pMold->ActInfo.ClampCls  = 0;

			pMold->Clamp.v_set  = 0;
			pMold->Clamp.p_set  = 0;

			pMold->Clamp.Step = 13000;
			break;

		/*-------------------------------------------------------------------------------*/
		/*-------------------------------- Clamp open  ----------------------------------*/
		/*-------------------------------------------------------------------------------*/
		case 10100: /* open delay*/
			if(pMold->TimeSet.ClampOpnDelay != 0)
			{
				pMold->Clamp.Timer.IN = 1;
				pMold->Clamp.Timer.PT = pMold->TimeSet.ClampOpnDelay;
				pMold->Clamp.Step 	  = 10200;

				//gExSPCS
				if(pMold == & LMold)
				{
					gExSPC[ExIndex].LMold.ClampOpnDelay = pMold->TimeSet.ClampOpnDelay/100.0;
				}
				else
				{
					gExSPC[ExIndex].RMold.ClampOpnDelay = pMold->TimeSet.ClampOpnDelay/100.0;
				}

			}
			else
			{
				pMold->Clamp.Step = 10300;
			}
			break;

		case 10200: /* delay ok */
			pMold->TimeDis.ClampOpnDelay = pMold->Clamp.Timer.ET;
			if (1 == pMold->Clamp.Timer.Q)
			{
				pMold->Clamp.Timer.IN        = 0;
				//	pMold->TimeDis.ClampOpnDelay = 0;
				pMold->Clamp.Step = 10300;
			}
			break;

		case 10300:	/* valve open delay  */
			if(0 == pMold->Clamp.OpnHWSwitch)
			{
				pMold->Clamp.rAfterPress2_Tolerance = (pClampFix->pPress2Hold/10) *0.2;
				if(pMold == &LMold)
				{
					pMold->Clamp.S_OpnSlowDrive  = xTogLinearLTrans(pClampPara->S_OpnSlow);
					pMold->Clamp.S_OpnEndDrive 	 = xTogLinearLTrans(pClampPara->S_OpnEnd);
				}
				else
				{
					pMold->Clamp.S_OpnSlowDrive  = xTogLinearRTrans(pClampPara->S_OpnSlow);
					pMold->Clamp.S_OpnEndDrive 	 = xTogLinearRTrans(pClampPara->S_OpnEnd);
				}

				pMold->Clamp.LimitTimer.IN = 1;
				if(1 == gMachineInfo.MachineReset)
					/*if(1 == gMachineInfo.MachineReset && 1 == gMachineInfo.Manual)*/  /* 自動復歸  */
				{
					pMold->Clamp.LimitTimer.PT = pMold->TimeSet.CycleAlarmTime;
				}
				else
				{
					pMold->Clamp.LimitTimer.PT = pMold->TimeSet.ClampOpnAlarmTime;
				}

				pMold->Clamp.vProfGen.Ts = tTask;
				pMold->Clamp.vProfGen.Tj = pClampFix->Open.Tj;
				pMold->Clamp.vProfGen.Td = pClampFix->Open.Td;

				pMold->Clamp.vProfGen.accel = pClampFix->Open.accel;
				if(pMold->Clamp.vProfGen.accel <= 0.0)pMold->Clamp.vProfGen.accel = 1000;

				pMold->Clamp.vProfGen.decel = pClampFix->Open.accel;
				if(pMold->Clamp.vProfGen.decel <= 0.0)pMold->Clamp.vProfGen.decel = 1000;

				pMold->Clamp.vProfGen.decel_end = pClampFix->Open.decel_end;
				if(pMold->Clamp.vProfGen.decel_end <= 0.0)pMold->Clamp.vProfGen.decel_end = 100;

				pMold->Clamp.vProfGen.v_start = 0.0;

				/*if(1 == gMachineInfo.MachineReset && 1 == gMachineInfo.Manual)*/  /* 自動復歸  */
				if(1 == gMachineInfo.MachineReset)
				{
//					pMold->Clamp.vProfGen.decel_end = 5.0 * pMold->Clamp.vProfGen.v_set;
					pMold->Clamp.vProfGen.decel_end = pClampFix->Open.decel_end;
					if(pMold->Clamp.vProfGen.decel_end <= 0.0)pMold->Clamp.vProfGen.decel_end = 100;

					pMold->Clamp.vProfGen.v_end	= 0;
					if(pMold->TimeSet.ClampLockTime == 0 )
					{
						pMold->Clamp.vProfGen.s_end = pMold->Clamp.S_OpnEndDrive;
					}
					else if(pMold->TimeSet.ClampLockTime != 0 )
					{
						pMold->Clamp.vProfGen.s_end = pMold->Clamp.S_OpnEndDrive + pMold->Clamp.rAfterPress2_Tolerance;
					}
					pMold->Clamp.vProfGen.init  = 1;
					pMold->Clamp.Step = 10420;

				}
				else if(1 == gMachineInfo.PinCalibration && 1 == gMachineInfo.Calib)
				{
					pMold->Clamp.vProfGen.decel_end = 5.0 * pMold->Clamp.vProfGen.v_set;
					if(pMold->Clamp.vProfGen.decel_end <= 0.0)pMold->Clamp.vProfGen.decel_end = 100;

					pMold->Clamp.vProfGen.v_end	= 0;
					if(pMold->TimeSet.ClampLockTime == 0 )
					{
						pMold->Clamp.vProfGen.s_end = pMold->Clamp.S_OpnEndDrive;
					}
					else if(pMold->TimeSet.ClampLockTime != 0 )
					{
						pMold->Clamp.vProfGen.s_end = pMold->Clamp.S_OpnEndDrive + pMold->Clamp.rAfterPress2_Tolerance;
					}
					pMold->Clamp.vProfGen.init  = 1;

					pMold->Clamp.Step = 10420;
				}
				else
				{
					if (pMold->Clamp.S_OpnSlow >0) //open slow
					{
						//						pMold->Clamp.vProfGen.v_end	= pMold->Clamp.V_Opn;
						//						pMold->Clamp.vProfGen.s_end = pMold->Clamp.S_OpnSlowDrive;
						//						pMold->Clamp.vProfGen.init  = 1;

						pMold->Clamp.vProfGen.v_end	= 0.0;
						if(pMold->TimeSet.ClampLockTime == 0 )
						{
							pMold->Clamp.vProfGen.s_end = pMold->Clamp.S_OpnEndDrive;
						}
						else if(pMold->TimeSet.ClampLockTime != 0 )
						{
							pMold->Clamp.vProfGen.s_end = pMold->Clamp.S_OpnEndDrive + pMold->Clamp.rAfterPress2_Tolerance;
						}
						pMold->Clamp.vProfGen.init  = 1;

						pMold->Clamp.Step = 10400;
					}
					else   					      //open quick
					{
						pMold->Clamp.vProfGen.v_end	= 0.0;
						if(pMold->TimeSet.ClampLockTime == 0 )
						{
							pMold->Clamp.vProfGen.s_end = pMold->Clamp.S_OpnEndDrive;
						}
						else if(pMold->TimeSet.ClampLockTime != 0 )
						{
							pMold->Clamp.vProfGen.s_end = pMold->Clamp.S_OpnEndDrive + pMold->Clamp.rAfterPress2_Tolerance;
						}
						pMold->Clamp.vProfGen.init  = 1;

						pMold->Clamp.Step = 10420;
					}
				}
			}
			else
			{
				pMold->HwAlarm.ClampOpnHWSwitch = 1;
				pMold->Clamp.Step = 41000;
			}
			break;

		case 10400:  /* open slow */
			pMold->ActInfo.ClampOpn  = 1;

			pMold->Clamp.vProfGen.v_set = pMold->Clamp.V_OpnSlow;

			/* call profile function */
			HydvProfGen(& pMold->Clamp.vProfGen);

			pMold->Clamp.p_set = pClampPara->P_OpnSlow;
			pMold->Clamp.v_set = pMold->Clamp.vProfGen.v_out;

			pMold->Clamp.actTjOpn = pMold->Clamp.vProfGen.Tj;

			/*  reached target position */
			if(pMold->Clamp.vProfGen.s_act >= pMold->Clamp.S_OpnSlowDrive)
			{
				//				pMold->Clamp.vProfGen.v_start = pMold->Clamp.v_set;
				//				pMold->Clamp.vProfGen.v_end	= 0.0;
				//				pMold->Clamp.vProfGen.s_end = pMold->Clamp.S_OpnEndDrive;
				//				pMold->Clamp.vProfGen.init  = 1;

				pMold->Clamp.Step = 10420;
			}

			if(1 == pMold->Clamp.OpnHWSwitch)
			{
				pMold->HwAlarm.ClampOpnHWSwitch = 1;
				pMold->Clamp.Step = 41000;
			}
			break;

		case 10420:  /* open quick  */
			pMold->ActInfo.ClampOpn  = 1;

			if(1 == gMachineInfo.MachineReset)
			{
				pMold->Clamp.vProfGen.v_set = pMold->Clamp.V_OpnReset;
				pMold->Clamp.p_set = pClampPara->P_OpnReset;
			}
			else
			{
				pMold->Clamp.vProfGen.v_set = pMold->Clamp.V_Opn;
				pMold->Clamp.p_set = pClampPara->P_Opn;;
			}

			/* call profile function */
			HydvProfGen(& pMold->Clamp.vProfGen);

			pMold->Clamp.v_set = pMold->Clamp.vProfGen.v_out;

			pMold->Clamp.actTjOpn = pMold->Clamp.vProfGen.Tj;

			/*  reached target position */
			if(pMold->Clamp.vProfGen.s_act >= pMold->Clamp.vProfGen.s_end - pMold->Clamp.Tolerance * Toggle_ToleranceFactor)
			{
				pMold->Clamp.v_set = 0;
				pMold->Clamp.Step = 10500;
			}

			if(1 == pMold->Clamp.OpnHWSwitch)
			{
				pMold->HwAlarm.ClampOpnHWSwitch = 1;
				pMold->Clamp.Step = 41000;
			}
			break;

		case 10500:
			if(1 == gMachineInfo.Auto)
			{
				pSPC->tCalmpOpn = pMold->Clamp.LimitTimer.ET/100.0;

				//gExSPC
				if(pMold == & LMold)
				{
					gExSPC[ExIndex].LMold.tClampOpn = pMold->Clamp.LimitTimer.ET/100.0;
				}
				else
				{
					gExSPC[ExIndex].RMold.tClampOpn = pMold->Clamp.LimitTimer.ET/100.0;
				}

			}
			pMold->Clamp.LimitTimer.IN = 0;

			pMold->Clamp.Step = 10600;
			//			if(pMold->ValveDelay.ClampOpn != 0)
			//			{
			//				pMold->Clamp.Timer.IN = 1;
			//				pMold->Clamp.Timer.PT = pMold->ValveDelay.ClampOpn;
			//				pMold->Clamp.Step = 10600;
			//			}
			//			else
			//			{
			//				pMold->Clamp.Step = 13000;
			//			}

			break;

		case 10600:

			pMold->Clamp.Timer.IN = 0;
			pMold->ActInfo.ClampOpn  = 0;
			pMold->ActInfo.ClampCls  = 0;

			pMold->Clamp.v_set  = 0;
			pMold->Clamp.p_set = 0;

			pMold->Clamp.Step = 13000;

			break;

		case 13000:
			break;

		/* --------------- 调校开模 --------------- */
		case 15000:
			if(0 == pMold->Clamp.OpnHWSwitch)
			{
				pMold->ActInfo.ClampOpn  = 1;

				pMold->Clamp.p_set = pClampFix->pCalibMax;
				pMold->Clamp.v_set = pClampFix->vCalibMax*10;

			}

			if(1 == pMold->Clamp.OpnHWSwitch)
			{
				pMold->HwAlarm.ClampOpnHWSwitch = 1;
				pMold->Clamp.Step = 41000;
			}
			break;

		/* ----------------------------  manual stop ------------------------- */
		case 20000:
			pMold->Clamp.Timer.IN      = 0;
			pMold->Clamp.LimitTimer.IN = 0;
			pMoldUser->Clamp.Timer.IN = 0;/*Albert*/

			pMold->ActInfo.ClampOpn = 0;
			pMold->ActInfo.ClampCls = 0;

			pMold->Clamp.p_old = pMold->Clamp.p_set;
			pMold->Clamp.Step = 21000;
			break;

		case 21000:
			pMold->Clamp.vRamp.Once = 0;
			pMold->Clamp.vRamp.Set = pMold->Clamp.v_set;

			pMold->Clamp.vRamp.Ts = tTask;

			if(pMold->Clamp.v_set > 0)
			{
				pMold->Clamp.vRamp.Accel = pClampFix->Open.accel_stop;
			}
			else
			{
				pMold->Clamp.vRamp.Accel = pClampFix->Close.accel_stop;
			}

			/* call profile function */
			HydSCurveRamp(&pMold->Clamp.vRamp);

			//	pMold->Clamp.p_set = 100.0;
			pMold->Clamp.v_set = pMold->Clamp.vRamp.Out;

			pMold->Clamp.Step = 22000;
			break;

		case 22000:
			pMold->Clamp.vRamp.Ts = tTask;
			pMold->Clamp.vRamp.Set = 0.0;

			/* call profile function */
			HydSCurveRamp(&pMold->Clamp.vRamp);

			pMold->Clamp.p_set = pMold->Clamp.p_old;
			pMold->Clamp.v_set = pMold->Clamp.vRamp.Out;

			if(pMold->Clamp.v_set < 0.1 && pMold->Clamp.v_set > -0.1)
			{
				pMold->Clamp.v_set = 0.0;
				pMold->Clamp.p_set =0;
				pMold->Clamp.Step = 0;

				pMold->Carriage.BtnOffDlyFlag = 1;  //owen Avoid Motor Fw/Bw quick switch
			}
			break;

		/* ----------------------------  Instance stop ------------------------- */
		case 30000:
			pMold->Clamp.Timer.IN      = 0;
			pMold->Clamp.LimitTimer.IN = 0;
			pMoldUser->Clamp.Timer.IN = 0;/*Albert*/

			pMold->ActInfo.ClampOpn = 0;
			pMold->ActInfo.ClampCls = 0;

			pMold->Clamp.vRamp.Once = 0;
			pMold->Clamp.vRamp.Set = pMold->Clamp.v_set;

			pMold->Clamp.vRamp.Ts = tTask;

			pMold->Clamp.vRamp.Accel = INSTANCY_STOP_ACCEL;

			/* call profile function */
			HydSCurveRamp(&pMold->Clamp.vRamp);

			//	pMold->Clamp.p_set = 100.0;
			pMold->Clamp.v_set = pMold->Clamp.vRamp.Out;

			pMold->Clamp.Step = 31000;
			break;

		case 31000:
			pMold->Clamp.vRamp.Ts = tTask;
			pMold->Clamp.vRamp.Set = 0.0;

			/* call profile function */
			HydSCurveRamp(&pMold->Clamp.vRamp);

			pMold->Clamp.p_set = pMold->Clamp.p_old;
			pMold->Clamp.v_set = pMold->Clamp.vRamp.Out;

			if(pMold->Clamp.v_set < 0.1 && pMold->Clamp.v_set > -0.1)
			{
				pMold->Clamp.v_set = 0.0;
				pMold->Clamp.p_set =0;
				pMold->Clamp.Step = 0;

				pMold->Carriage.BtnOffDlyFlag = 1;  //owen Avoid Motor Fw/Bw quick switch
			}
			break;

		/* ----------------------------  Error step ------------------------- */
		case 40000:
			pMold->Clamp.Timer.IN      = 0;
			pMold->Clamp.LimitTimer.IN = 0;

			pMold->ActInfo.ClampOpn = 0;
			pMold->ActInfo.ClampCls = 0;

			pMold->Clamp.v_set = 0.0;
			pMold->Clamp.p_set =0;

			break;

		/* ----------------------------  auto run stop ------------------------- */
		case 41000:
			pMold->Clamp.Timer.IN      = 0;
			pMold->Clamp.LimitTimer.IN = 0;

			pMold->ActInfo.ClampOpn = 0;
			pMold->ActInfo.ClampCls = 0;

			pMold->Clamp.Step = 42000;
			break;

		case 42000:
			pMold->Clamp.vRamp.Internal.Once = 0;
			pMold->Clamp.vRamp.Set = pMold->Clamp.v_set;

			pMold->Clamp.vRamp.Ts = tTask;

			pMold->Clamp.vRamp.Accel = INSTANCY_STOP_ACCEL;

			/* call profile function */
			HydSCurveRamp(&pMold->Clamp.vRamp);
			pMold->Clamp.Step = 43000;
			break;

		case 43000:
			pMold->Clamp.vRamp.Ts = tTask;
			pMold->Clamp.vRamp.Set = 0.0;

			/* call profile function */
			HydSCurveRamp(&pMold->Clamp.vRamp);

			//	pMold->Clamp.p_set = 100.0;
			pMold->Clamp.v_set = pMold->Clamp.vRamp.Out;

			if(pMold->Clamp.v_set < 0.1 && pMold->Clamp.v_set > -0.1)
			{
				pMold->Clamp.p_set =0;
				pMold->Clamp.v_set = 0.0;
				pMold->Clamp.Step = 40000;
			}
			break;
	}/* end of switch */

	if(pMold->Clamp.Step > 300 && pMold->Clamp.Step  < 800)
	{
		pMold->TimeDis.ClampClsAlarmTime = pMold->Clamp.LimitTimer.ET;
	}
	else if(pMold->Clamp.Step > 10300 && pMold->Clamp.Step  < 10800)
	{
		pMold->TimeDis.ClampOpnAlarmTime = pMold->Clamp.LimitTimer.ET;
	}

	/* ----------------- clamp open / close timeout --------------------  */
	if(1 == pMold->Clamp.LimitTimer.Q && 1 == gMachineInfo.TimeLimit)
	{
		if(pMold->Clamp.Step < 4000 && pMold->Clamp.Step > 200)		/* clamp close  */
		{
			pMold->Alarm.ClampNotAtClsDI = 1;
		}

		if(pMold->Clamp.Step < 13000 && pMold->Clamp.Step > 10200)	/* clamp open  */
		{
			pMold->Alarm.ClampNotAtOpnDI = 1;
		}

		pMold->Clamp.LimitTimer.IN = 0;
		pMold->Clamp.Step = 41000;
	}

	/* ----------------- clamp open / close action limit --------------------  */

	if(pMold->Clamp.Step < 3000 && pMold->Clamp.Step > 200) 	/* clamp close  */
	{

		if( 0 == pMold->TransDIn.SubMoldClsLimit)
		{
			pMold->Alarm.SubMoldNotAtOpnPos  = !pMold->TransDIn.SubMoldOpnLimit;
			pMold->Clamp.Step = 41000;
		}

		if( 0 == pMold->TransDIn.BottomSubMoldClsLimit)
		{
			pMold->Alarm.SubMoldNotAtOpnPos  = !pMold->TransDIn.BottomSubMoldClsLimit;
			pMold->Clamp.Step = 41000;
		}

		if(1 == gMachineInfo.Auto && 1 == gMachineFix.Option.bCoolPinUpNextCycClampCls)   /* 特殊模式  "於下一循環關模後轉一上"  */
		{
//			if ( 0 == pMold->TransDIn.CoolPin2UpLimit || 0 == pMold->TransDIn.CoolPin3UpLimit )
//			{
//				pMold->Alarm.CoolPin2NotAtUpPos = !pMold->TransDIn.CoolPin2UpLimit;
//				pMold->Alarm.CoolPin3NotAtUpPos	= !pMold->TransDIn.CoolPin3UpLimit;
//				pMold->Clamp.Step = 41000;
//			}
		}
		else
		{
			if (0 == pMold->TransDIn.CoolPinUpLimit )
			{
				pMold->Alarm.CoolPinNotAtUpPos	= !pMold->TransDIn.CoolPinUpLimit;
				pMold->Clamp.Step = 41000;
			}

		}

		if(0 == gMachineInfo.Auto)
		{
			if(0 == pMold->Robot.Transfer.BwPos)
			{
				pMold->Alarm.RobotNotAtBwPos = !pMold->Robot.Transfer.BwPos;
				pMold->Clamp.Step = 41000;
			}
		}

		if(1 == gMachineInfo.Auto )
		{
			if(0 == pMold->Carriage.FwPos)
			{
				pMold->Alarm.CarriageNotAtFwDI  = !pMold->Carriage.FwPos;
				pMold->Clamp.Step = 41000;
			}
		}

		/* 模内吹针在回位   */
		//      if(0 == pMold->TransDIn.InnerPinBwLimit)
		//      {
		//         pMold->Alarm.InnerPinNotAtBwPos = !pMold->TransDIn.InnerPinBwLimit;
		//         pMold->Clamp.Step = 41000;
		//      }

		//      if(1 == gMachineInfo.TimeLimit)
		//      {
		//         if(0 == pMold->Carriage.FwPos)
		//         {
		//            pMold->Alarm.CarriageNotAtFwDI  = !pMold->Carriage.FwPos;
		//            pMold->Clamp.Step = 41000;
		//         }
		//      }
		//      else
		//      {
		//         if(0 == pMold->Carriage.BwPos
		//			&& 0 == pMold->Carriage.FwPos
		//			&& 0 == pMold->BlowPin.UpPos)
		//         {
		//         	pMold->Alarm.CarriageNotAtBwDI = !pMold->Carriage.BwPos;
		//         	pMold->Alarm.BlowPinNotAtUpPos = !pMold->BlowPin.UpPos;
		//         	pMold->Clamp.Step = 41000;
		//         }
		//      }/* if(1 == gMachineInfo.Manual) */
	}/* if(pMold->Clamp.Step < 3000 && pMold->Clamp.Step > 200) */

	if(pMold->Clamp.Step < 13000 && pMold->Clamp.Step > 10200)  /* clamp open  */
	{

		/* 切飞边非退位  */
		if( 0 == pMold->TransDIn.TopDeflashBwLimit )
		{
			pMold->Alarm.TopDeflashNotAtBwPos = !pMold->TransDIn.TopDeflashBwLimit;
			pMold->Clamp.Step = 41000;
		}

		if( 0 == pMold->TransDIn.BottomDeflashBwLimit)
		{
			pMold->Alarm.BottomDeflashNotAtBwPos = !pMold->TransDIn.BottomDeflashBwLimit;
			pMold->Clamp.Step = 41000;
		}

		if(0 == gMachineInfo.Auto)
		{
			if(0 == pMold->TransDIn.ExtRobotUpLmit )
			{
				pMold->Alarm.ExtRobotNotAtUp = !pMold->TransDIn.ExtRobotUpLmit;
				pMold->Clamp.Step = 41000;
			}
		}

	}/* if(pMold->Clamp.Step < 13000 && pMold->Clamp.Step > 10200) */

	//	if((13000 >= pMold->Clamp.Step) && (10200 < pMold->Clamp.Step))
	//	{
	//		if(pMold == &RMold)
	//		{
	//			RobotClampTime.IN = pMold->Clamp.OpnPos;/*Albert RobotClampOpn*/
	//			RobotClampTime.PT = RobotClampTimePara;
	//		}
	//		if(pMold == & LMold)
	//		{
	//			LRobotClampTime.IN = pMold->Clamp.OpnPos;
	//			LRobotClampTime.PT = LRobotClampTimePara;
	//		}
	//	}
	//	else
	//	{
	////		RobotClampTime.IN = 0;/*Albert RobotClampOpn*/
	//	}
	//	if(pMold == &RMold)
	//	{
	//		if(RobotClampTime.Q)
	//		{
	//			RobotClampTime.IN = 0;
	//		}
	//		pMold->ValveOut.RobotClampOpn = RobotClampTime.Q;
	//
	//	}
	//	if(pMold == &LMold)
	//	{
	//		if(LRobotClampTime.Q)
	//		{
	//			LRobotClampTime.IN = 0;
	//		}
	//		pMold->ValveOut.RobotClampOpn = LRobotClampTime.Q;
	//	}

}/*end of function */

REAL xTogLinearLTrans(REAL pClampPos)
{
	xTogLinearL.Y = pClampPos;
	HydLinear(&xTogLinearL);
	if(0 == xTogLinearL.status)
	{
		return xTogLinearL.X;
	}
	else
	{
		return 0;
	}
}

REAL xTogLinearRTrans(REAL pClampPos)
{
	xTogLinearR.Y = pClampPos;
	HydLinear(&xTogLinearR);
	if(0 == xTogLinearR.status)
	{
		return xTogLinearR.X;
	}
	else
	{
		return 0;
	}
}

void ButtonOffDelay(Mold_typ * pMold,timer_typ * pTimer)
{
	if(  1 == pMold->Clamp.BtnOffDlyFlag )
	{
		pTimer->IN = 1;
		pTimer->PT = 200;

		if( 1 == pTimer->Q)
		{
			pMold->Clamp.BtnOffDlyFlag = 0;
		}
	}
	else
	{
		pTimer->IN = 0;
	}

}
```

#### clamp.var
```iecst
VAR
	ValveDelay : REAL;
	tTask : REAL := 0.0;
	tErrorDelay : REAL;
	rMin : REAL;
	RTInfo_Task : RTInfo := (0);
	vActHydDT2_L : HydDT2;
	vActHydDT2_R : HydDT2;
	ToggleInputL : USINT;
	ToggleInputR : USINT;
	ToggleLOld : ARRAY[0..30] OF Hyd_Node_typ;
	ToggleROld : ARRAY[0..30] OF Hyd_Node_typ;
	TogLinearL : HydLinear;
	TogLinearR : HydLinear;
	xToggleNodeL : ARRAY[0..30] OF Hyd_Node_typ;
	xTogLinearL : HydLinear;
	xToggleNodeR : ARRAY[0..30] OF Hyd_Node_typ;
	xTogLinearR : HydLinear;
	bToggle_Init : USINT;
	oldToggleLinNodeNum : USINT;
	ToggleLinNodeNum : USINT;
END_VAR
(*For robot singal stand on timer*)
VAR
	OldRClampOpnDI : USINT;
	OldLClampOpnDI : USINT;
	bClampPropValveOutputInverse : USINT;
	Toggle_ToleranceFactor : REAL := 1;
END_VAR
(*Test*)
VAR
	Test_vTimeProf_accel : REAL := 1000;
	Test_vTimeProf_decel : REAL := 1000;
END_VAR
(*ExtInMoldSticker*)
VAR
	OldRExtInMoldStickerBwLimit : USINT;
	OldLExtInMoldStickerBwLimit : USINT;
END_VAR
```

### Program Logical/process/tonnage (ANSIC, version 1.00.0) - lock mold

#### tonnage.c
```c
/********************************************************************
 * COPYRIGHT --  B&R China
 ********************************************************************
 * Program: Tonnage
 * File: Tonnage.c
 * Author: lijianjun
 * Created: March 06, 2013
 ********************************************************************
 * Implementation of program Tonnage --- mold Tonnage
 ********************************************************************/

#include <bur/plctypes.h>

#ifdef _DEFAULT_INCLUDES
#include <AsDefault.h>
#endif

/**************************************************************************************
                            Function Declarations
**************************************************************************************/

void Lock( Mold_typ * pMold,Clamp_Para_typ * pClampPara);

/**************************************************************************************
     	        		I N I T U P  O F   T H E   T A S K
**************************************************************************************/
_INIT void init ( void )
{
	LMold.Lock.Step = 30000;
	RMold.Lock.Step = 30000;
} /* end of _INIT */

 /*************************************************************************************
        				C Y C L I C   P A R T   O F   T H E   T A S K
**************************************************************************************/

_CYCLIC void cyclic ( void )
{

	Lock(&LMold,&gMachinePara.MoldL.Clamp);
	Lock(&RMold,&gMachinePara.MoldR.Clamp);

	gMachineOut.LMold.ClampLocking = LMold.ValveOut.Lock;
	gMachineOut.RMold.ClampLocking = RMold.ValveOut.Lock;

	gMachineOut.LMold.ClampClsAux  = LMold.ValveOut.ClampClsAux;
	gMachineOut.RMold.ClampClsAux  = RMold.ValveOut.ClampClsAux;

} /* end of _CYCLIC */

void Lock( Mold_typ * pMold,Clamp_Para_typ * pClampPara)
{

	switch ( pMold->Lock.Step )
	{
		/*------------------ stop all the output ------------------*/
		case 0:
			pMold->Lock.Timer.IN = 0;

			if(pMold->Clamp.Step <= 300 && pMold->Clamp.Step >= 500 )  // Clamp Close Fast Do not Close valve
			{
				pMold->ValveOut.Lock = 0;		/*Clamp Locking valve*/
				pMold->ValveOut.ClampClsAux = 0;/*Clamp Close aux. valve*/
			}

			break;

		/*------------------ Lock  -------------------- */
		case 100: 	/* delay */

			if(pMold->TimeSet.ClampLockDly != 0)
			{
				pMold->Lock.Timer.IN = 1;
				pMold->Lock.Timer.PT = pMold->TimeSet.ClampLockDly;
				pMold->Lock.Step = 200;
			}
			else
			{
				pMold->Lock.Step = 300;
			}

			break;

		case 200: 	/* locking delay */

			pMold->ValveOut.Lock = 0;		/*Clamp Locking valve*/
			pMold->ValveOut.ClampClsAux = 0;/*Clamp Close aux. valve*/

			pMold->TimeDis.ClampLockDly = pMold->Lock.Timer.ET;
			if (1 == pMold->Lock.Timer.Q)
			{
				pMold->Lock.Timer.IN = 0;
				pMold->TimeDis.ClampLockDly = 0;
				pMold->Lock.Step = 300;
			}
			break;

		case 300: 	/* set lock time */

			if(pMold->TimeSet.ClampLockTime != 0)
			{
				pMold->Lock.Timer.IN = 1;
				pMold->Lock.Timer.PT = pMold->TimeSet.ClampLockTime;
				pMold->Lock.Step = 400;
			}
			else
			{
				pMold->Lock.Step = 500;
			}

			break;

		case 400: 	/* locking */

			pMold->ValveOut.Lock = 1;		/*Clamp Locking valve*/
			pMold->ValveOut.ClampClsAux = 1;/*Clamp Close aux. valve*/

			//			pMold->Lock.p_set = pClampPara->P_Tonnage;
			//			pMold->Lock.v_set = pClampPara->V_Tonnage;

			pMold->TimeDis.ClampLockTime = pMold->Lock.Timer.ET;
			if (1 == pMold->Lock.Timer.Q)
			{
				pMold->Lock.Timer.IN = 0;
				//	pMold->TimeDis.ClampLockTime = 0;

				pMold->ValveOut.Lock = 0;		/*Clamp Locking valve*/
				pMold->ValveOut.ClampClsAux = 0;/*Clamp Close aux. valve*/

				//				pMold->Lock.p_set = 0.0;
				//				pMold->Lock.v_set = 0.0;

				pMold->Lock.Step = 500;
			}
			break;

		case 500:

			pMold->ValveOut.Lock = 0;		/*Clamp Locking valve*/
			pMold->ValveOut.ClampClsAux = 0;/*Clamp Close aux. valve*/

			pMold->Lock.Timer.IN = 0;
			pMold->Lock.Step = 3000;
			break;

		case 3000:
			break;

		case 10100:

			pMold->Lock.Step = 13000;
			break;

		case 13000:
			break;

		/*--------------- Manual action stop -----------------*/
		case 20000:
			pMold->ValveOut.Lock = 0;		/*Clamp Locking valve*/
			pMold->ValveOut.ClampClsAux = 0;/*Clamp Close aux. valve*/

			pMold->Lock.p_set = 0.0;
			pMold->Lock.v_set = 0.0;

			pMold->Lock.Timer.IN         = 0;
			//   pMold->TimeDis.ClampLockTime = 0;
			pMold->Lock.Step = 0;
			break;

		/*--------------- Instance stop -----------------*/
		case 30000:
			pMold->ValveOut.Lock = 0;		/*Clamp Locking valve*/
			pMold->ValveOut.ClampClsAux = 0;/*Clamp Close aux. valve*/

			pMold->Lock.p_set = 0.0;
			pMold->Lock.v_set = 0.0;

			pMold->Lock.Timer.IN = 0;
			//	pMold->TimeDis.ClampLockTime = 0;
			pMold->Lock.Step = 0;

			break;
	}/* end of switch */

	//	pMold->Lock.aoPropValve = (INT)(pMold->Lock.v_set * 327.67);

}/*end of function */
```

### Program Logical/process/support (ANSIC, version 1.00.0) - air support

#### supportair.c
```c
/********************************************************************
 * COPYRIGHT --  B&R China
 ********************************************************************
 * Program: Supportair
 * File: Supportair.c
 * Author: lijianjun
 * Created: March 06, 2013
 ********************************************************************
 * Implementation of program Supportair --- Supportair
 ********************************************************************/

#include <bur/plctypes.h>

#ifdef _DEFAULT_INCLUDES
	#include <AsDefault.h>
#endif

/**************************************************************************************
                            Function Declarations
**************************************************************************************/
//void SupportAir( Mold_typ * pMold,Support_Para_typ * pSupportPara);
void SupportAir( Mold_typ * pMold,Support_Para_typ * pSupportPara,Mold_Para_User_typ * pMoldUser);
void SupportAir_Time( Mold_typ * pMold,Support_Para_typ * pSupportPara,Mold_Para_User_typ * pMoldUser,Support_Fix_typ * pSupportFix);
void SupportSuckAir_Time( Mold_typ * pMold,Support_Para_typ * pSupportPara,Mold_Para_User_typ * pMoldUser);
/**************************************************************************************
     	        		I N I T U P  O F   T H E   T A S K
**************************************************************************************/
_INIT void init ( void )
 {
	RTInfo_Task.enable = 1;
	RTInfo(&RTInfo_Task);

	tTask = RTInfo_Task.cycle_time/1000.0/1000.0;		/*  from us ---> s  */
 } /* end of _INIT */

 /*************************************************************************************
        				C Y C L I C   P A R T   O F   T H E   T A S K
**************************************************************************************/

 _CYCLIC void cyclic ( void )
 {
	gMachinePara.SupportAirEnable[0] =0;  //ipis0305
	gMachinePara.SupportAirEnable[1] =0;

	if(gUserPara.FluxSensor[0].Zero < 0.1)gUserPara.FluxSensor[0].Zero = 1.0;
	if(gUserPara.FluxSensor[0].Max < 0.1 )gUserPara.FluxSensor[0].Max  = 8.0;
	if(gUserPara.FluxSensor[0].Length < 0.1 )gUserPara.FluxSensor[0].Length = 80.0;

	if(gUserPara.FluxSensor[0].Max - gUserPara.FluxSensor[0].Zero > 0.0)
	{
		RMold.SupportAir.FlowDieA = (RMold.SupportAir.aiFlowDieA - gUserPara.FluxSensor[0].Zero * 3726.7) * gUserPara.FluxSensor[0].Length /
			                         (gUserPara.FluxSensor[0].Max * 3276.7 - gUserPara.FluxSensor[0].Zero * 3276.7);
	}
	else
	{
		RMold.SupportAir.FlowDieA = 0.0;
	}

	LMold.SupportAir.FlowDieA = RMold.SupportAir.FlowDieA;

	if(gUserPara.FluxSensor[1].Zero < 0.1)gUserPara.FluxSensor[1].Zero = 1.0;
	if(gUserPara.FluxSensor[1].Max < 0.1 )gUserPara.FluxSensor[1].Max  = 8.0;
	if(gUserPara.FluxSensor[1].Length < 0.1 )gUserPara.FluxSensor[1].Length = 80.0;

	if(gUserPara.FluxSensor[1].Max - gUserPara.FluxSensor[1].Zero > 0.0)
	{
		RMold.SupportAir.FlowDieB = (RMold.SupportAir.aiFlowDieB - gUserPara.FluxSensor[1].Zero * 3726.7) * gUserPara.FluxSensor[1].Length /
			                         (gUserPara.FluxSensor[2].Max * 3276.7 - gUserPara.FluxSensor[2].Zero * 3276.7);
	}
	else
	{
		RMold.SupportAir.FlowDieB = 0.0;
	}

	LMold.SupportAir.FlowDieB = RMold.SupportAir.FlowDieB;

	if(gUserPara.FluxSensor[2].Zero < 0.1)gUserPara.FluxSensor[2].Zero = 1.0;
	if(gUserPara.FluxSensor[2].Max < 0.1 )gUserPara.FluxSensor[2].Max  = 8.0;
	if(gUserPara.FluxSensor[2].Length < 0.1 )gUserPara.FluxSensor[2].Length = 80.0;

	if(gUserPara.FluxSensor[2].Max - gUserPara.FluxSensor[2].Zero != 0.0)
	{
		RMold.SupportAir.FlowDieC = (RMold.SupportAir.aiFlowDieC - gUserPara.FluxSensor[2].Zero * 3726.7) * gUserPara.FluxSensor[2].Length /
			                         (gUserPara.FluxSensor[2].Max * 3276.7 - gUserPara.FluxSensor[2].Zero * 3276.7);
	}
	else
	{
		RMold.SupportAir.FlowDieC = 0.0;
	}

	LMold.SupportAir.FlowDieB = RMold.SupportAir.FlowDieB;

	if(gUserPara.FluxSensor[3].Zero < 0.1)gUserPara.FluxSensor[3].Zero = 1.0;
	if(gUserPara.FluxSensor[3].Max < 0.1 )gUserPara.FluxSensor[3].Max  = 8.0;
	if(gUserPara.FluxSensor[3].Length < 0.1 )gUserPara.FluxSensor[3].Length = 80.0;

	if(gUserPara.FluxSensor[3].Max - gUserPara.FluxSensor[3].Zero != 0.0)
	{
		RMold.SupportAir.FlowDieD = (RMold.SupportAir.aiFlowDieD - gUserPara.FluxSensor[3].Zero * 3726.7) * gUserPara.FluxSensor[3].Length /
			                         (gUserPara.FluxSensor[3].Max * 3276.7 - gUserPara.FluxSensor[3].Zero * 3276.7);
	}
	else
	{
		RMold.SupportAir.FlowDieD = 0.0;
	}

	LMold.SupportAir.FlowDieD = RMold.SupportAir.FlowDieD;

//	SupportAir(&LMold, &gMachinePara.MoldL.SupportAir,&gUserPara.LMold);
//	SupportAir(&RMold, &gMachinePara.MoldR.SupportAir,&gUserPara.RMold);

	/*------------- SupportAirMode--------------- */
	gMachineFix.MoldL.SupportAir.eSupportAirMode = gMachineFix.MoldR.SupportAir.eSupportAirMode;

	SupportAir_Time(&LMold, &gMachinePara.MoldL.SupportAir,&gUserPara.LMold,&gMachinePara.MoldL.SupportAir);
	SupportAir_Time(&RMold, &gMachinePara.MoldR.SupportAir,&gUserPara.RMold,&gMachinePara.MoldR.SupportAir);

	SupportSuckAir_Time(&LMold, &gMachinePara.MoldL.SupportAir,&gUserPara.LMold);
	SupportSuckAir_Time(&RMold, &gMachinePara.MoldR.SupportAir,&gUserPara.RMold);

	if(1 == gMachineInfo.Auto)
	{
		gMachineOut.SupportAir_1 = LMold.SupportAir.Out_1 | RMold.SupportAir.Out_1;
		gMachineOut.SupportAir_2 = LMold.SupportAir.Out_2 | RMold.SupportAir.Out_2;

		/*----------------------------------------------------*/
		/*-------------------Left side------------------------*/
		/*----------------------------------------------------*/

		if(gThickProf.TimSet.CycleTime != 0)
		{
			/*Albert Start count calculate left*/
			switch (uCntStepL)
			{
				case 0:/*weit step*/
					if(LMold.SupportAir.cntTime > 0)
					{
						if(tTask != 0)
						{
							uCntTimeL = LMold.SupportAir.cntTime/100/tTask;
							uCntStepL = 1;
						}

					}
					break;
				case 1:/*Start count, since tTask is 4ms so If we need s counting should chagne the counter*/
					if(uCntTimeL > 0)
					{
						uCntTimeL -= tTask;
					}
					else
					{
						LMold.SupportAir.cntTime = 0;
						uCntTimeL = 0;
						uCntStepL = 0;
					}

					break;
			}
			//	Make this time from 100ms to 1000ms
			//					|						Make this time from s to 1000ms
			//					|									|			Change to %
			//					|									|				|			dvide by gThickProf cycleTime 100ms
			//					|									|				|					|
			idxThickL = ((gThickProf.TimSet.CycleTime*10) - (uCntTimeL*tTask*1000))*10/gThickProf.TimSet.CycleTime;
			nCurrentPointL = (INT)idxThickL;/*Albert*/

			/*----------------------------------------------------*/
			/*-------------------Right side------------------------*/
			/*----------------------------------------------------*/
			switch (uCntStepR)
			{
				case 0:/*weit step*/
					if(RMold.SupportAir.cntTime > 0)
					{
						if(tTask != 0)
						{
							uCntTimeR = (REAL)RMold.SupportAir.cntTime/100/tTask;
							uCntStepR = 1;
						}
					}
					break;
				case 1:/*Start count, since tTask is 4ms so If we need s counting should chagne the counter*/
					if(uCntTimeR > 0)
					{
						uCntTimeR-=tTask;
					}
					else
					{
						RMold.SupportAir.cntTime = 0;
						uCntTimeR = 0;
						uCntStepR = 0;
					}
					break;
			}
			//	Make this time from 100ms to 1000ms
			//					|						Make this time from s to 1000ms
			//					|									|			Change to %
			//					|									|				|			dvide by gThickProf cycleTime 100ms
			//					|									|				|					|
			idxThickR = ((gThickProf.TimSet.CycleTime*10) - (uCntTimeR*tTask*1000))*10/gThickProf.TimSet.CycleTime;
			nCurrentPointR = (INT)idxThickR;/*Albert*/
		}
	}
	else
	{
		gMachineOut.SupportAir_1 = 0;
		gMachineOut.SupportAir_2 = 0;

		LMold.SupportAir.PressureSet = 0.0;

		LMold.SupportAir.FlowSetDieA = 0.0;
		LMold.SupportAir.FlowSetDieB = 0.0;
		LMold.SupportAir.FlowSetDieC = 0.0;
		LMold.SupportAir.FlowSetDieD = 0.0;

		RMold.SupportAir.PressureSet = 0.0;

		RMold.SupportAir.FlowSetDieA = 0.0;
		RMold.SupportAir.FlowSetDieB = 0.0;
		RMold.SupportAir.FlowSetDieC = 0.0;
		RMold.SupportAir.FlowSetDieD = 0.0;

		if(gThickProf.TimSet.CycleTime != 0)
		{
			/*----------------------------------------------------*/
			/*-------------------Left side------------------------*/
			/*----------------------------------------------------*/

			/*Albert Start count calculate left*/
			switch (uCntStepL)
			{
				case 0:/*weit step*/

					if(LMold.SupportAir.cntTime > 0)
					{
						if(tTask != 0)
						{
							uCntTimeL = LMold.SupportAir.cntTime/100/tTask;
							uCntStepL = 1;
						}

					}

					break;
				case 1:/*Start count, since tTask is 4ms so If we need s counting should chagne the counter*/
					if(uCntTimeL > 0)
					{
						uCntTimeL -= tTask;
					}
					else
					{
						LMold.SupportAir.cntTime = 0;
						uCntTimeL = 0;
						uCntStepL = 0;
					}

					break;
			}
			//	Make this time from 100ms to 1000ms
			//					|						Make this time from s to 1000ms
			//					|									|			Change to %
			//					|									|				|			dvide by gThickProf cycleTime 100ms
			//					|									|				|					|
			idxThickL = ((gThickProf.TimSet.CycleTime*10) - (uCntTimeL*tTask*1000))*10/gThickProf.TimSet.CycleTime;

//			if(LMold.SupportAir.cntTime > 0)LMold.SupportAir.cntTime--;
//			idxThickL = (gThickProf.TimSet.CycleTime - LMold.SupportAir.cntTime)*100.0/gThickProf.TimSet.CycleTime;
//			idxThickL = gThickData.CurrentTime * 100.0/gThickProf.TimSet.CycleTime;/*Albert*/
			nCurrentPointL = (INT)idxThickL;/*Albert*/

			if(idxThickL > LMold.TimeSet.SupportAirStart[0] && idxThickL < LMold.TimeSet.SupportAirStop[0])
			{
				if(gMachinePara.SupportAirEnable[0])
				{
					gMachineOut.SupportAir_1 = 1;

					LMold.SupportAir.PressureSet = gMachinePara.MoldL.SupportAir.SetPre_1;

					LMold.SupportAir.FlowSetDieA = gMachinePara.MoldL.SupportAir.SetFlowA1;
					LMold.SupportAir.FlowSetDieB = gMachinePara.MoldL.SupportAir.SetFlowB1;
					LMold.SupportAir.FlowSetDieC = gMachinePara.MoldL.SupportAir.SetFlowC1;
					LMold.SupportAir.FlowSetDieD = gMachinePara.MoldL.SupportAir.SetFlowD1;
				}
			}
			else if(idxThickL > LMold.TimeSet.SupportAirStart[1] && idxThickL < LMold.TimeSet.SupportAirStop[1])
			{
				if(gMachinePara.SupportAirEnable[1])
				{
					gMachineOut.SupportAir_2 = 1;

					LMold.SupportAir.PressureSet = gMachinePara.MoldL.SupportAir.SetPre_1;

					LMold.SupportAir.FlowSetDieA = gMachinePara.MoldL.SupportAir.SetFlowA2;
					LMold.SupportAir.FlowSetDieB = gMachinePara.MoldL.SupportAir.SetFlowB2;
					LMold.SupportAir.FlowSetDieC = gMachinePara.MoldL.SupportAir.SetFlowC2;
					LMold.SupportAir.FlowSetDieD = gMachinePara.MoldL.SupportAir.SetFlowD2;
				}
			}

			/*----------------------------------------------------*/
			/*-------------------Right side------------------------*/
			/*----------------------------------------------------*/

			/*Albert Start count calculate right*/
			switch (uCntStepR)
			{
				case 0:/*weit step*/

					if(RMold.SupportAir.cntTime > 0)
					{
						if(tTask != 0)
						{
							uCntTimeR = (REAL)RMold.SupportAir.cntTime/100/tTask;
							uCntStepR = 1;
						}
					}

					break;
				case 1:/*Start count, since tTask is 4ms so If we need s counting should chagne the counter*/
					if(uCntTimeR > 0)
					{
						uCntTimeR-=tTask;
					}
					else
					{
						RMold.SupportAir.cntTime = 0;
						uCntTimeR = 0;
						uCntStepR = 0;
					}

					break;
			}

//			if(RMold.SupportAir.cntTime > 0) /*RMold.SupportAir.cntTime-=tTask;*/

			//	Make this time from 100ms to 1000ms
			//					|						Make this time from s to 1000ms
			//					|									|			Change to %
			//					|									|				|			dvide by gThickProf cycleTime 100ms
			//					|									|				|					|
			idxThickR = ((gThickProf.TimSet.CycleTime*10) - (uCntTimeR*tTask*1000))*10/gThickProf.TimSet.CycleTime;
//			idxThickR = (gThickProf.TimSet.CycleTime - RMold.SupportAir.cntTime)*100.0/gThickProf.TimSet.CycleTime;
//			idxThickR = gThickData.CurrentTime * 100.0/gThickProf.TimSet.CycleTime;/*Albert*/
			nCurrentPointR = (INT)idxThickR;/*Albert*/

			if(idxThickR > RMold.TimeSet.SupportAirStart[0] && idxThickR < RMold.TimeSet.SupportAirStop[0])
			{
				if(gMachinePara.SupportAirEnable[0])
				{
					gMachineOut.SupportAir_1 = 1;

					RMold.SupportAir.PressureSet = gMachinePara.MoldR.SupportAir.SetPre_1;

					RMold.SupportAir.FlowSetDieA = gMachinePara.MoldR.SupportAir.SetFlowA1;
					RMold.SupportAir.FlowSetDieB = gMachinePara.MoldR.SupportAir.SetFlowB1;
					RMold.SupportAir.FlowSetDieC = gMachinePara.MoldR.SupportAir.SetFlowC1;
					RMold.SupportAir.FlowSetDieD = gMachinePara.MoldR.SupportAir.SetFlowD1;
				}
			}
			else if(idxThickR > RMold.TimeSet.SupportAirStart[1] && idxThickR < RMold.TimeSet.SupportAirStop[1])
			{
				if(gMachinePara.SupportAirEnable[1])
				{
					gMachineOut.SupportAir_2 = 1;

					RMold.SupportAir.PressureSet = gMachinePara.MoldR.SupportAir.SetPre_2;

					RMold.SupportAir.FlowSetDieA = gMachinePara.MoldR.SupportAir.SetFlowA2;
					RMold.SupportAir.FlowSetDieB = gMachinePara.MoldR.SupportAir.SetFlowB2;
					RMold.SupportAir.FlowSetDieC = gMachinePara.MoldR.SupportAir.SetFlowC2;
					RMold.SupportAir.FlowSetDieD = gMachinePara.MoldR.SupportAir.SetFlowD2;
				}
			}

//			if(1 == gMachinePara.SupportAirVentEnable)
//			{
//				if((gMachinePara.SupportAirVentingStrart == idxThickL) || (gMachinePara.SupportAirVentingStrart == idxThickR))
//				{
//					RMold.SupportAir.Step = 200;
//				}
//			}
		}

//		if(1 == bTestButton && gMachineInfo.Auto != 1)
//		{
//			gMachineOut.SupportAir_1 = 1;
//
//			gMachineOut.SuckAir_1 = 1;
//
//			RMold.SupportAir.PressureSet = gMachinePara.MoldR.SupportAir.SetPre_1;
//
//			RMold.SupportAir.FlowSetDieA = gMachinePara.MoldR.SupportAir.SetFlowA1;
//			RMold.SupportAir.FlowSetDieB = gMachinePara.MoldR.SupportAir.SetFlowB1;
//			RMold.SupportAir.FlowSetDieC = gMachinePara.MoldR.SupportAir.SetFlowC1;
//			RMold.SupportAir.FlowSetDieD = gMachinePara.MoldR.SupportAir.SetFlowD1;
//		}

//		if(0 == bTestButton && gMachineInfo.Auto != 1)
//		{
//			gMachineOut.SuckAir_1 = 0;
//		}
	}
	//SupportAir_TimeVersion(脹風)
	gMachineOut.SupportAir_TimeVersion 		= (LMold.ValveOut.SupportAir_TimeVersion| RMold.ValveOut.SupportAir_TimeVersion);

	//SuckAir_TimeVersion(模頭抽真空)
	gMachineOut.SuckAir_TimeVersion 		= (LMold.ValveOut.SuckAir_TimeVersion| RMold.ValveOut.SuckAir_TimeVersion);
	gMachineOut.SuckAirRelieve_TimeVersion	= (LMold.ValveOut.SuckAirRelieve_TimeVersion| RMold.ValveOut.SupportAir_TimeVersion);

	gUserPara.LMold.TimeSet.SupportAirSecDelay = gUserPara.RMold.TimeSet.SupportAirSecDelay;
	gUserPara.LMold.TimeSet.SupportAirSecTime = gUserPara.RMold.TimeSet.SupportAirSecTime;

}/* end of _CYCLIC */

void SupportAir( Mold_typ * pMold, Support_Para_typ * pSupportPara, Mold_Para_User_typ * pMoldUser)
{
	/* ---------------- 模頭吹風 --------------------- */

	/*Albert, use nCurrentPoint get actual thick data*/
//	if(gMachineInfo.Auto == 1)
//	{
//		if(pMold == &RMold)
//		{
//			nCurrentPointR = gThickData.FocusNum;/*Albert*/
//		}
//
//		if(pMold == &LMold)
//		{
//			nCurrentPointL = gThickData.FocusNum;/*Albert*/
//		}
//	}

	if(1 == pMold->OnceSupport)
	{
		pMold->SupportAir.Out_1 = 0;
		pMold->SupportAir.Out_2 = 0;

		pMold->SupportAir.PressureSet = 0.0;

		pMold->SupportAir.FlowSetDieA = 0.0;
		pMold->SupportAir.FlowSetDieB = 0.0;
		pMold->SupportAir.FlowSetDieC = 0.0;
		pMold->SupportAir.FlowSetDieD = 0.0;

		if(gThickData.FocusNum > pMold->TimeSet.SupportAirStart[0] &&
	 	   gThickData.FocusNum < pMold->TimeSet.SupportAirStop[0])
	 	{
			if(gMachinePara.SupportAirEnable[0])
			{
				pMold->SupportAir.Out_1 = 1;

				pMold->SupportAir.PressureSet = pSupportPara->SetPre_1;

				pMold->SupportAir.FlowSetDieA = pSupportPara->SetFlowA1;
				pMold->SupportAir.FlowSetDieB = pSupportPara->SetFlowB1;
				pMold->SupportAir.FlowSetDieC = pSupportPara->SetFlowC1;
				pMold->SupportAir.FlowSetDieD = pSupportPara->SetFlowD1;
			}
		}
		else if(gThickData.FocusNum > pMold->TimeSet.SupportAirStart[1]&&
	 	   	  gThickData.FocusNum < pMold->TimeSet.SupportAirStop[1])
		{
			if(gMachinePara.SupportAirEnable[1])
			{
				pMold->SupportAir.Out_2 = 1;

				pMold->SupportAir.PressureSet = pSupportPara->SetPre_2;

				pMold->SupportAir.FlowSetDieA = pSupportPara->SetFlowA2;
				pMold->SupportAir.FlowSetDieB = pSupportPara->SetFlowB2;
				pMold->SupportAir.FlowSetDieC = pSupportPara->SetFlowC2;
				pMold->SupportAir.FlowSetDieD = pSupportPara->SetFlowD2;
			}
		}/* else if */
	}

	if(99 == gThickData.FocusNum)
	{
		pMold->OnceSupport = 0;
	}

	if(0 == gMachineInfo.Auto)
	{
		pMold->OnceSupport = 0;
		pMold->SupportAir.Out_1 = 0;
		pMold->SupportAir.Out_2 = 0;
	}

	/*  模頭排氣/吸氣  */
	if(pMold == &RMold)
	{
		switch(pMold->SupportAir.Step)
		{
			case 100:
				if(1 == gMachinePara.SupportAirVentEnable)
				{
//					if(gThickData.FocusNum == gMachinePara.SupportAirVentingStrart)
//					{
						gMachineOut.SuckAir_1 = 0;
						gMachineOut.SuckAir_2 = 0;
						pMold->SupportAir.Timer.IN = 0;
						pMold->SupportAir.Step = 200;	/*   排气启动   */
//					}
				}
				else
				{
					pMold->SupportAir.Step = 3000;
				}
				break;

			case 200:
				gMachineOut.SuckAir_1 = 0;
				gMachineOut.SuckAir_2 = 0;
				pMold->SupportAir.Timer.IN = 0;

				if(gMachinePara.SupportAirVentingDelay != 0)
				{
					pMold->SupportAir.Step = 300;
				}
				else
				{
					pMold->SupportAir.Step = 500;
				}
				break;

			case 300:
				pMold->SupportAir.Timer.IN = 1;
				pMold->SupportAir.Timer.PT = gMachinePara.SupportAirVentingDelay;
				pMold->SupportAir.Step = 400;
				break;

			case 400:
				SuckAirDelayDis = pMold->SupportAir.Timer.ET;
				if(1 == pMold->SupportAir.Timer.Q)
				{
					pMold->SupportAir.Timer.IN = 0;
				//	SuckAirDelayDis = 0;
					pMold->SupportAir.Step = 500;
				}
				break;

			case 500:
				if(gMachinePara.SupportAirVentingTime != 0)
				{
					pMold->SupportAir.Step = 600;
				}
				else
				{
					pMold->SupportAir.Timer.IN = 0;
			//		pMold->SupportAir.Step = 3000;
				pMold->SupportAir.Step = 800; //20190130 ipis
				}
				break;

			case 600:
				pMold->SupportAir.Timer.IN = 1;
				pMold->SupportAir.Timer.PT = gMachinePara.SupportAirVentingTime;
				pMold->SupportAir.Step = 700;
				break;

			case 700:
				gMachineOut.SuckAir_1 = 1;
				gMachineOut.SuckAir_2 = 1;
				SuckAirTimeDis = pMold->SupportAir.Timer.ET;
				if(1 == pMold->SupportAir.Timer.Q)
				{
					gMachineOut.SuckAir_1 = 0;
					gMachineOut.SuckAir_2 = 0;
					pMold->SupportAir.Timer.IN = 0;
			//		SuckAirTimeDis = 0;
					pMold->SupportAir.Step = 800;
				}
				break;

			case 800:/*Start second suckair delay time*/

				if(pMoldUser->TimeSet.SupportAirSecDelay != 0)
				{
					pMold->SupportAir.Timer.IN = 1;
					pMold->SupportAir.Timer.PT = pMoldUser->TimeSet.SupportAirSecDelay;
					pMold->SupportAir.Step = 900;
				}
				else
				{
					pMold->SupportAir.Step = 1000;
				}
				break;
			case 900:
				gMachineOut.SuckAir_1 = 0;
				gMachineOut.SuckAir_2 = 0;

				pMoldUser->TimeDis.SupportAirSecDelay= pMold->SupportAir.Timer.ET;
				if(pMold->SupportAir.Timer.Q)
				{
					pMold->SupportAir.Timer.IN = 0;
					pMold->SupportAir.Step = 1000;
				}
				break;

			case 1000:/*Start Second Support air time*/

				if(pMoldUser->TimeSet.SupportAirSecTime != 0)
				{
					pMold->SupportAir.Timer.IN = 1;
					pMold->SupportAir.Timer.PT = pMoldUser->TimeSet.SupportAirSecTime;
					pMold->SupportAir.Step = 1100;
				}
				else
				{
					pMold->SupportAir.Step = 3000;
				}
				break;

			case 1100:
				gMachineOut.SuckAir_1 = 1;
				gMachineOut.SuckAir_2 = 1;

				pMoldUser->TimeDis.SupportAirSecTime = pMold->SupportAir.Timer.ET;

				if(pMold->SupportAir.Timer.Q)
				{
					pMold->SupportAir.Timer.IN = 0;
					pMold->SupportAir.Step = 3000;
				}

				break;

			case 3000:
				gMachineOut.SuckAir_1 = 0;
				gMachineOut.SuckAir_2 = 0;
				pMold->SupportAir.Timer.IN = 0;

//				if(1 == gMachineInfo.Auto)
//				{
//					pMold->SupportAir.Step = 100;
//				}
//				else
//				{
//					pMold->SupportAir.Step = 0;
//				}
				break;

			case 20000:
				gMachineOut.SupportAir_1 = 0;
				gMachineOut.SuckAir_1  = 0;
				gMachineOut.SuckAir_2  = 0;

				pMold->SupportAir.Timer.IN = 0;
				SuckAirDelayDis = 0;
				SuckAirTimeDis  = 0;

				pMold->SupportAir.Step = 0;
				break;

			case 30000:
				gMachineOut.SupportAir_1 = 0;
				gMachineOut.SuckAir_1  = 0;
				gMachineOut.SuckAir_2  = 0;

				pMold->SupportAir.Timer.IN = 0;
				SuckAirDelayDis = 0;
				SuckAirTimeDis  = 0;

				pMold->SupportAir.Step = 0;
				break;
		}/* switch(SuckAirStep) */
	 }
 }

void SupportAir_Time( Mold_typ * pMold,Support_Para_typ * pSupportPara,Mold_Para_User_typ * pMoldUser,Support_Fix_typ * pSupportFix)
{
	/* ---------------- 模頭漲風  時間版本  --------------------- */
	switch(pMold->SupportAir.Step)
	{
		case 0:
			pMold->ValveOut.SupportAir_TimeVersion = 0;

			pMold->SupportAir.Timer.IN = 0;

			break;

		case 100:
			if(1 == gMachinePara.SupportAirTimeVersionEnable)
			{
				pMold->ValveOut.SupportAir_TimeVersion = 0;
				pMold->SupportAir.Timer.IN = 0;
				pMold->SupportAir.Step = 200;	/*   排气启动   */
			}
			else
			{
				pMold->SupportAir.Step = 3000;
			}
			break;

		case 200: /*Start first suport air delay time*/
			pMold->ValveOut.SupportAir_TimeVersion = 0;
			pMold->SupportAir.Timer.IN = 0;

			if(pMold->TimeSet.SupportAirDelay)
			{
				pMold->SupportAir.Step = 300;
			}
			else
			{
				pMold->SupportAir.Step = 500;
			}
			break;

		case 300:
			pMold->SupportAir.Timer.IN = 1;
			pMold->SupportAir.Timer.PT = pMold->TimeSet.SupportAirDelay;
			pMold->SupportAir.Step = 400;
			break;

		case 400:
			pMold->TimeDis.SupportAirDelay = pMold->SupportAir.Timer.ET;
			if(1 == pMold->SupportAir.Timer.Q)
			{
				pMold->SupportAir.Timer.IN = 0;
				pMold->SupportAir.Step = 500;
			}
			break;

		case 500: /*Start first suport air time*/
			if(pMold->TimeSet.SupportAirTime != 0)
			{
				pMold->SupportAir.Step = 600;
			}
			else
			{
				pMold->SupportAir.Timer.IN = 0;
				pMold->SupportAir.Step = 800;
			}
			break;

		case 600:
			pMold->SupportAir.Timer.IN = 1;
			pMold->SupportAir.Timer.PT = pMold->TimeSet.SupportAirTime;
			pMold->SupportAir.Step = 700;

			break;

		case 700:
			pMold->ValveOut.SupportAir_TimeVersion = 1;
			pMold->TimeDis.SupportAirTime = pMold->SupportAir.Timer.ET;

			if(1 == pMold->SupportAir.Timer.Q)
			{
				pMold->ValveOut.SupportAir_TimeVersion = 0;
				pMold->SupportAir.Timer.IN = 0;

				if( SUPPORTAIR_MODE_STANDARD == pSupportFix->eSupportAirMode)
				{
					pMold->SupportAir.Step = 800;
				}
				else if(SUPPORTAIR_MODE_AFTER_CLAMP_CLS == pSupportFix->eSupportAirMode)
				{
					pMold->SupportAir.Step = 3000;  // only one time support air
				}
			}
			break;

		case 800:/*Start second suport air delay time*/

			if(pMold->TimeSet.SupportAirSecDelay != 0)
			{
				pMold->SupportAir.Timer.IN = 1;
				pMold->SupportAir.Timer.PT = pMold->TimeSet.SupportAirSecDelay;
				pMold->SupportAir.Step = 900;
			}
			else
			{
				pMold->SupportAir.Step = 1000;
			}
			break;
		case 900:
			pMold->ValveOut.SupportAir_TimeVersion = 0;
			pMold->TimeDis.SupportAirSecDelay = pMold->SupportAir.Timer.ET;
			if(pMold->SupportAir.Timer.Q)
			{
				pMold->SupportAir.Timer.IN = 0;
				pMold->SupportAir.Step = 1000;
			}
			break;

		case 1000:/*Start Second Support air time*/

			if(pMold->TimeSet.SupportAirSecTime != 0)
			{
				pMold->SupportAir.Timer.IN = 1;
				pMold->SupportAir.Timer.PT = pMold->TimeSet.SupportAirSecTime;
				pMold->SupportAir.Step = 1100;
			}
			else
			{
				pMold->SupportAir.Step = 3000;
			}
			break;

		case 1100:
			pMold->ValveOut.SupportAir_TimeVersion = 1;
			pMold->TimeDis.SupportAirSecTime = pMold->SupportAir.Timer.ET;

			if(pMold->SupportAir.Timer.Q)
			{
				pMold->SupportAir.Timer.IN = 0;
				pMold->SupportAir.Step = 3000;
			}

			break;

		case 3000:
			pMold->ValveOut.SupportAir_TimeVersion = 0;
			pMold->SupportAir.Timer.IN = 0;

			//				if(1 == gMachineInfo.Auto)
			//				{
			//					pMold->SupportAir.Step = 100;
			//				}
			//				else
			//				{
			//					pMold->SupportAir.Step = 0;
			//				}
			break;

		case 20000:
			pMold->ValveOut.SupportAir_TimeVersion = 0;
			pMold->SupportAir.Timer.IN = 0;
			pMold->SupportAir.Step = 0;

			break;

		case 30000:
			pMold->ValveOut.SupportAir_TimeVersion = 0;
			pMold->SupportAir.Timer.IN = 0;
			pMold->SupportAir.Step = 0;

			break;
	}/* switch(SupportAir) */

}

void SupportSuckAir_Time( Mold_typ * pMold, Support_Para_typ * pSupportPara, Mold_Para_User_typ * pMoldUser)
{
	/* ---------------- 模頭抽真空  時間版本  --------------------- */
	switch(pMold->SupportSuckAir.Step)
	{
		case 0:
			pMold->ValveOut.SuckAir_TimeVersion = 0;
			pMold->ValveOut.SuckAirRelieve_TimeVersion = 0;
			pMold->SupportSuckAir.Timer.IN = 0;

			break;

		case 100:
			if(1 == gUserPara.SupportAirVentTimeVersionEnable)
			{
				pMold->ValveOut.SuckAir_TimeVersion = 0;
				pMold->ValveOut.SuckAirRelieve_TimeVersion = 0;
				pMold->SupportSuckAir.Timer.IN = 0;
				pMold->SupportSuckAir.Step = 200;	/*   吸氣启动   */
			}
			else
			{
				pMold->SupportSuckAir.Step = 3000;
			}
			break;

		case 200:
			pMold->ValveOut.SuckAir_TimeVersion = 0;
			pMold->ValveOut.SuckAirRelieve_TimeVersion = 0;
			pMold->SupportSuckAir.Timer.IN = 0;

			if(gMachinePara.SupportAirVentingDelay != 0)
			{
				pMold->SupportSuckAir.Step = 300;
			}
			else
			{
				pMold->SupportSuckAir.Step = 500;
			}
			break;

		case 300:
			pMold->SupportSuckAir.Timer.IN = 1;
			pMold->SupportSuckAir.Timer.PT = gMachinePara.SupportAirVentingDelay;
			pMold->SupportSuckAir.Step = 400;
			break;

		case 400:   // SupportAirVenting  Delay
			SuckAirDelayDis = pMold->SupportSuckAir.Timer.ET;
			if(1 == pMold->SupportSuckAir.Timer.Q)
			{
				pMold->SupportSuckAir.Timer.IN = 0;
//				SuckAirDelayDis = 0;
				pMold->SupportSuckAir.Step = 500;
			}
			break;

		case 500:
			if(gMachinePara.SupportAirVentingTime != 0)
			{
				pMold->SupportSuckAir.Step = 600;
			}
			else
			{
				pMold->SupportSuckAir.Timer.IN = 0;
				pMold->SupportSuckAir.Step = 3000;
			}
			break;

		case 600:
			pMold->SupportSuckAir.Timer.IN = 1;
			pMold->SupportSuckAir.Timer.PT = gMachinePara.SupportAirVentingTime;
			pMold->SupportSuckAir.Step = 700;

			break;

		case 700:    //SupportAirVenting Time
			pMold->ValveOut.SuckAir_TimeVersion = 1;
			pMold->ValveOut.SuckAirRelieve_TimeVersion = 1;
			SuckAirTimeDis = pMold->SupportSuckAir.Timer.ET;
			if(1 == pMold->SupportSuckAir.Timer.Q)
			{
				pMold->ValveOut.SuckAir_TimeVersion = 0;
				pMold->ValveOut.SuckAirRelieve_TimeVersion = 0;
				pMold->SupportSuckAir.Timer.IN = 0;
//				SuckAirTimeDis = 0;
				pMold->SupportSuckAir.Step = 3000;
			}
			break;

		case 3000:
			pMold->ValveOut.SuckAir_TimeVersion = 0;
			pMold->ValveOut.SuckAirRelieve_TimeVersion = 0;
			pMold->SupportSuckAir.Timer.IN = 0;

			break;

		case 20000:
			pMold->ValveOut.SuckAir_TimeVersion = 0;
			pMold->ValveOut.SuckAirRelieve_TimeVersion = 0;
			pMold->SupportSuckAir.Timer.IN = 0;
			pMold->SupportSuckAir.Step = 0;

			break;

		case 30000:
			pMold->ValveOut.SuckAir_TimeVersion = 0;
			pMold->ValveOut.SuckAirRelieve_TimeVersion = 0;
			pMold->SupportSuckAir.Timer.IN = 0;
			pMold->SupportSuckAir.Step = 0;

			break;
	}/* switch(SupportSuckAir) */

}
```

#### support.var
```iecst
VAR
	bTestButton : BOOL;
	idxThickL : REAL;
	idxThickR : REAL;
	SuckAirDelayDis : UDINT;
	SuckAirTimeDis : UDINT;
	nCurrentPointL : INT;
	nCurrentPointR : INT;
END_VAR
(*Cycle Time*)
VAR
	tTask : REAL := 0.0;
	RTInfo_Task : RTInfo := (0);
	uCntTimeR_TON_10ms : TON_10ms;
	uCntTimeL_TON_10ms : TON_10ms;
	uCntTimeR : UDINT;
	uCntTimeL : UDINT;
	uCntStepR : USINT;
	uCntStepL : USINT;
END_VAR
```

### Program Logical/process/blowpin (ANSIC, version 1.00.0) - blow pin
